LIN {X 0,Y 340.654,Z 947.959,A -85,B 0,C 180,E1 16403.067,E2 16403.067} C_VEL
LIN {X 0,Y 348.105,Z 969.694,A -85,B 0,C 180,E1 16408.833,E2 16408.833} C_VEL
LIN {X 0,Y 350.733,Z 979.844,A -85,B 0,C 180,E1 16411.083,E2 16411.083} C_VEL
LIN {X 0,Y 337.341,Z 1017.391,A -85,B 0,C 180,E1 16414.207,E2 16414.207} C_VEL
LIN {X 0,Y 321.586,Z 1053.328,A -85,B 0,C 180,E1 16418.46,E2 16418.46} C_VEL
LIN {X 0,Y 305.489,Z 1085.768,A -85,B 0,C 180,E1 16424.011,E2 16424.011} C_VEL
LIN {X 0,Y 291.393,Z 1112.806,A -85,B 0,C 180,E1 16430.628,E2 16430.628} C_VEL
LIN {X 0,Y 280.047,Z 1134.815,A -85,B 0,C 180,E1 16438.272,E2 16438.272} C_VEL
LIN {X 0,Y 272.429,Z 1152.316,A -85,B 0,C 180,E1 16447.187,E2 16447.187} C_VEL
LIN {X 0,Y 269.212,Z 1162.751,A -85,B 0,C 180,E1 16455.39,E2 16455.39} C_VEL
LIN {X 0,Y 268.092,Z 1168.645,A -85,B 0,C 180,E1 16463.537,E2 16463.537} C_VEL
LIN {X 0,Y 268.297,Z 1170.082,A -85,B 0,C 180,E1 16470,E2 16470} C_VEL
LIN {X 0,Y 268.113,Z 1168.65,A -85,B 0,C 180,E1 16476.464,E2 16476.464} C_VEL
LIN {X 0,Y 269.134,Z 1162.757,A -85,B 0,C 180,E1 16484.615,E2 16484.615} C_VEL
LIN {X 0,Y 272.422,Z 1152.335,A -85,B 0,C 180,E1 16492.815,E2 16492.815} C_VEL
LIN {X 0,Y 280.074,Z 1134.846,A -85,B 0,C 180,E1 16501.724,E2 16501.724} C_VEL
LIN {X 0,Y 292.426,Z 1110.76,A -85,B 0,C 180,E1 16509.976,E2 16509.976} C_VEL
LIN {X 0,Y 307.416,Z 1082.201,A -85,B 0,C 180,E1 16516.713,E2 16516.713} C_VEL
LIN {X 0,Y 323.735,Z 1049.016,A -85,B 0,C 180,E1 16522.139,E2 16522.139} C_VEL
LIN {X 0,Y 339.489,Z 1012.268,A -85,B 0,C 180,E1 16526.294,E2 16526.294} C_VEL
LIN {X 0,Y 350.803,Z 979.89,A -85,B 0,C 180,E1 16528.924,E2 16528.924} C_VEL
LIN {X 0,Y 344.157,Z 957.095,A -85,B 0,C 180,E1 16534.344,E2 16534.344} C_VEL
LIN {X 0,Y 344.02,Z 956.717,A -85,B 0,C 180,E1 16534.444,E2 16534.444} C_VEL
LIN {X 0,Y 340.378,Z 952.198,A -85,B 0,C 180,E1 16536.416,E2 16536.416} C_VEL
LIN {X 0,Y 333.985,Z 946.963,A -85,B 0,C 180,E1 16539.918,E2 16539.918} C_VEL
LIN {X 0,Y 328.108,Z 933.13,A -85,B 0,C 180,E1 16545.812,E2 16545.812} C_VEL
LIN {X 0,Y 324.423,Z 925.798,A -85,B 0,C 180,E1 16550.715,E2 16550.715} C_VEL
LIN {X 0,Y 322.252,Z 920.268,A -85,B 0,C 180,E1 16555.972,E2 16555.972} C_VEL
LIN {X 0,Y 322.042,Z 920.226,A -85,B 0,C 180,E1 16564.703,E2 16564.703} C_VEL
LIN {X 0,Y 324.764,Z 927.987,A -85,B 0,C 180,E1 16571.677,E2 16571.677} C_VEL
LIN {X 0,Y 328.984,Z 938.356,A -85,B 0,C 180,E1 16577.355,E2 16577.355} C_VEL
LIN {X 0,Y 334.486,Z 953.605,A -85,B 0,C 180,E1 16583.249,E2 16583.249} C_VEL
LIN {X 0,Y 339.367,Z 971.623,A -85,B 0,C 180,E1 16588.478,E2 16588.478} C_VEL
LIN {X 0,Y 341.727,Z 984.521,A -85,B 0,C 180,E1 16591.625,E2 16591.625} C_VEL
LIN {X 0,Y 326.648,Z 1021.482,A -85,B 0,C 180,E1 16595.426,E2 16595.426} C_VEL
LIN {X 0,Y 310.779,Z 1053.687,A -85,B 0,C 180,E1 16600.114,E2 16600.114} C_VEL
LIN {X 0,Y 295.445,Z 1081.297,A -85,B 0,C 180,E1 16605.785,E2 16605.785} C_VEL
LIN {X 0,Y 281.431,Z 1105.448,A -85,B 0,C 180,E1 16612.899,E2 16612.899} C_VEL
LIN {X 0,Y 270.826,Z 1124.108,A -85,B 0,C 180,E1 16620.821,E2 16620.821} C_VEL
LIN {X 0,Y 263.998,Z 1138.31,A -85,B 0,C 180,E1 16629.942,E2 16629.942} C_VEL
LIN {X 0,Y 261.06,Z 1146.198,A -85,B 0,C 180,E1 16638.325,E2 16638.325} C_VEL
LIN {X 0,Y 260.252,Z 1149.946,A -85,B 0,C 180,E1 16646.676,E2 16646.676} C_VEL
LIN {X 0,Y 260.353,Z 1149.923,A -85,B 0,C 180,E1 16653.322,E2 16653.322} C_VEL
LIN {X 0,Y 261.09,Z 1146.107,A -85,B 0,C 180,E1 16661.701,E2 16661.701} C_VEL
LIN {X 0,Y 264.034,Z 1138.177,A -85,B 0,C 180,E1 16670.054,E2 16670.054} C_VEL
LIN {X 0,Y 270.935,Z 1123.932,A -85,B 0,C 180,E1 16679.166,E2 16679.166} C_VEL
LIN {X 0,Y 282.862,Z 1103.055,A -85,B 0,C 180,E1 16687.843,E2 16687.843} C_VEL
LIN {X 0,Y 297.942,Z 1076.932,A -85,B 0,C 180,E1 16695.159,E2 16695.159} C_VEL
LIN {X 0,Y 314.902,Z 1045.612,A -85,B 0,C 180,E1 16701.132,E2 16701.132} C_VEL
LIN {X 0,Y 331.218,Z 1011.108,A -85,B 0,C 180,E1 16705.666,E2 16705.666} C_VEL
LIN {X 0,Y 341.719,Z 984.7,A -85,B 0,C 180,E1 16708.217,E2 16708.217} C_VEL
LIN {X 0,Y 337.435,Z 964.238,A -85,B 0,C 180,E1 16713.437,E2 16713.437} C_VEL
LIN {X 0,Y 331.773,Z 945.868,A -85,B 0,C 180,E1 16719.361,E2 16719.361} C_VEL
LIN {X 0,Y 326.407,Z 931.853,A -85,B 0,C 180,E1 16725.665,E2 16725.665} C_VEL
LIN {X 0,Y 323.079,Z 924.574,A -85,B 0,C 180,E1 16730.998,E2 16730.998} C_VEL
LIN {X 0,Y 322.055,Z 920.268,A -85,B 0,C 180,E1 16734.623,E2 16734.623} C_VEL
LIN {X 0,Y 321.831,Z 919.955,A -85,B 0,C 180,E1 16743.36,E2 16743.36} C_VEL
LIN {X 0,Y 322.694,Z 921.542,A -85,B 0,C 180,E1 16745.907,E2 16745.907} C_VEL
LIN {X 0,Y 325.815,Z 928.749,A -85,B 0,C 180,E1 16751.564,E2 16751.564} C_VEL
LIN {X 0,Y 330.368,Z 938.469,A -85,B 0,C 180,E1 16756.775,E2 16756.775} C_VEL
LIN {X 0,Y 337.309,Z 955.675,A -85,B 0,C 180,E1 16763.044,E2 16763.044} C_VEL
LIN {X 0,Y 343.984,Z 977.436,A -85,B 0,C 180,E1 16768.852,E2 16768.852} C_VEL
LIN {X 0,Y 345.164,Z 984.629,A -85,B 0,C 180,E1 16770.348,E2 16770.348} C_VEL
LIN {X 0,Y 330.908,Z 1021.712,A -85,B 0,C 180,E1 16773.523,E2 16773.523} C_VEL
LIN {X 0,Y 314.982,Z 1056.2,A -85,B 0,C 180,E1 16777.77,E2 16777.77} C_VEL
LIN {X 0,Y 298.773,Z 1087.349,A -85,B 0,C 180,E1 16783.282,E2 16783.282} C_VEL
LIN {X 0,Y 284.328,Z 1113.711,A -85,B 0,C 180,E1 16789.946,E2 16789.946} C_VEL
LIN {X 0,Y 272.063,Z 1136.394,A -85,B 0,C 180,E1 16798.203,E2 16798.203} C_VEL
LIN {X 0,Y 264.38,Z 1153.254,A -85,B 0,C 180,E1 16807.34,E2 16807.34} C_VEL
LIN {X 0,Y 261.037,Z 1164.056,A -85,B 0,C 180,E1 16816.631,E2 16816.631} C_VEL
LIN {X 0,Y 260.187,Z 1168.346,A -85,B 0,C 180,E1 16823.339,E2 16823.339} C_VEL
LIN {X 0,Y 260.397,Z 1169.786,A -85,B 0,C 180,E1 16830,E2 16830} C_VEL
LIN {X 0,Y 260.207,Z 1168.351,A -85,B 0,C 180,E1 16836.661,E2 16836.661} C_VEL
LIN {X 0,Y 261.337,Z 1162.455,A -85,B 0,C 180,E1 16845.061,E2 16845.061} C_VEL
LIN {X 0,Y 264.897,Z 1152.029,A -85,B 0,C 180,E1 16853.501,E2 16853.501} C_VEL
LIN {X 0,Y 273.056,Z 1134.611,A -85,B 0,C 180,E1 16862.604,E2 16862.604} C_VEL
LIN {X 0,Y 285.699,Z 1111.26,A -85,B 0,C 180,E1 16870.816,E2 16870.816} C_VEL
LIN {X 0,Y 301.193,Z 1083.104,A -85,B 0,C 180,E1 16877.62,E2 16877.62} C_VEL
LIN {X 0,Y 318.243,Z 1049.873,A -85,B 0,C 180,E1 16883.146,E2 16883.146} C_VEL
LIN {X 0,Y 334.398,Z 1013.673,A -85,B 0,C 180,E1 16887.292,E2 16887.292} C_VEL
LIN {X 0,Y 345.374,Z 983.208,A -85,B 0,C 180,E1 16889.856,E2 16889.856} C_VEL
LIN {X 0,Y 339.297,Z 961.193,A -85,B 0,C 180,E1 16895.359,E2 16895.359} C_VEL
LIN {X 0,Y 333.985,Z 946.963,A -85,B 0,C 180,E1 16899.918,E2 16899.918} C_VEL
LIN {X 0,Y 330.79,Z 943.941,A -85,B 0,C 180,E1 16902.054,E2 16902.054} C_VEL
LIN {X 0,Y 325.406,Z 941.02,A -85,B 0,C 180,E1 16905.775,E2 16905.775} C_VEL
LIN {X 0,Y 322.278,Z 933.67,A -85,B 0,C 180,E1 16910.228,E2 16910.228} C_VEL
LIN {X 0,Y 320.307,Z 928.989,A -85,B 0,C 180,E1 16914.593,E2 16914.593} C_VEL
LIN {X 0,Y 319.155,Z 927.085,A -85,B 0,C 180,E1 16920,E2 16920} C_VEL
LIN {X 0,Y 319.864,Z 928.113,A -85,B 0,C 180,E1 16925.414,E2 16925.414} C_VEL
LIN {X 0,Y 322.655,Z 937.222,A -85,B 0,C 180,E1 16932.637,E2 16932.637} C_VEL
LIN {X 0,Y 327.152,Z 949.317,A -85,B 0,C 180,E1 16938.836,E2 16938.836} C_VEL
LIN {X 0,Y 331.99,Z 965.451,A -85,B 0,C 180,E1 16944.622,E2 16944.622} C_VEL
LIN {X 0,Y 336.018,Z 985.699,A -85,B 0,C 180,E1 16950.157,E2 16950.157} C_VEL
LIN {X 0,Y 336.292,Z 988.923,A -85,B 0,C 180,E1 16950.887,E2 16950.887} C_VEL
LIN {X 0,Y 319.803,Z 1026.489,A -85,B 0,C 180,E1 16954.833,E2 16954.833} C_VEL
LIN {X 0,Y 303.201,Z 1058.494,A -85,B 0,C 180,E1 16959.741,E2 16959.741} C_VEL
LIN {X 0,Y 286.434,Z 1087.183,A -85,B 0,C 180,E1 16966.094,E2 16966.094} C_VEL
LIN {X 0,Y 271.46,Z 1111.385,A -85,B 0,C 180,E1 16973.971,E2 16973.971} C_VEL
LIN {X 0,Y 260.716,Z 1129.921,A -85,B 0,C 180,E1 16983.107,E2 16983.107} C_VEL
LIN {X 0,Y 254.827,Z 1142.335,A -85,B 0,C 180,E1 16992.777,E2 16992.777} C_VEL
LIN {X 0,Y 252.919,Z 1147.644,A -85,B 0,C 180,E1 16999.689,E2 16999.689} C_VEL
LIN {X 0,Y 252.363,Z 1150.242,A -85,B 0,C 180,E1 17006.572,E2 17006.572} C_VEL
LIN {X 0,Y 252.455,Z 1150.22,A -85,B 0,C 180,E1 17013.426,E2 17013.426} C_VEL
LIN {X 0,Y 253.258,Z 1146.428,A -85,B 0,C 180,E1 17022.037,E2 17022.037} C_VEL
LIN {X 0,Y 256.456,Z 1138.482,A -85,B 0,C 180,E1 17030.673,E2 17030.673} C_VEL
LIN {X 0,Y 263.849,Z 1124.239,A -85,B 0,C 180,E1 17040.028,E2 17040.028} C_VEL
LIN {X 0,Y 276.468,Z 1103.363,A -85,B 0,C 180,E1 17048.88,E2 17048.88} C_VEL
LIN {X 0,Y 292.297,Z 1077.238,A -85,B 0,C 180,E1 17056.283,E2 17056.283} C_VEL
LIN {X 0,Y 309.42,Z 1046.841,A -85,B 0,C 180,E1 17062.155,E2 17062.155} C_VEL
LIN {X 0,Y 326.738,Z 1011.505,A -85,B 0,C 180,E1 17066.813,E2 17066.813} C_VEL
LIN {X 0,Y 336.383,Z 988.492,A -85,B 0,C 180,E1 17069.046,E2 17069.046} C_VEL
LIN {X 0,Y 332.457,Z 968.245,A -85,B 0,C 180,E1 17074.459,E2 17074.459} C_VEL
LIN {X 0,Y 327.465,Z 950.69,A -85,B 0,C 180,E1 17080.484,E2 17080.484} C_VEL
LIN {X 0,Y 323.03,Z 938.176,A -85,B 0,C 180,E1 17086.493,E2 17086.493} C_VEL
LIN {X 0,Y 320.756,Z 932.535,A -85,B 0,C 180,E1 17090.525,E2 17090.525} C_VEL
LIN {X 0,Y 319.702,Z 927.802,A -85,B 0,C 180,E1 17094.584,E2 17094.584} C_VEL
LIN {X 0,Y 319.375,Z 927.351,A -85,B 0,C 180,E1 17102.708,E2 17102.708} C_VEL
LIN {X 0,Y 320.38,Z 929.773,A -85,B 0,C 180,E1 17106.276,E2 17106.276} C_VEL
LIN {X 0,Y 323.432,Z 937.155,A -85,B 0,C 180,E1 17111.983,E2 17111.983} C_VEL
LIN {X 0,Y 328.649,Z 949.187,A -85,B 0,C 180,E1 17118.055,E2 17118.055} C_VEL
LIN {X 0,Y 334.692,Z 966.317,A -85,B 0,C 180,E1 17123.939,E2 17123.939} C_VEL
LIN {X 0,Y 339.971,Z 986.661,A -85,B 0,C 180,E1 17129.225,E2 17129.225} C_VEL
LIN {X 0,Y 323.818,Z 1027.577,A -85,B 0,C 180,E1 17132.986,E2 17132.986} C_VEL
LIN {X 0,Y 306.824,Z 1062.218,A -85,B 0,C 180,E1 17137.528,E2 17137.528} C_VEL
LIN {X 0,Y 289.537,Z 1093.548,A -85,B 0,C 180,E1 17143.538,E2 17143.538} C_VEL
LIN {X 0,Y 273.838,Z 1120.582,A -85,B 0,C 180,E1 17151.154,E2 17151.154} C_VEL
LIN {X 0,Y 262.582,Z 1140.908,A -85,B 0,C 180,E1 17159.541,E2 17159.541} C_VEL
LIN {X 0,Y 255.421,Z 1156.492,A -85,B 0,C 180,E1 17169.239,E2 17169.239} C_VEL
LIN {X 0,Y 252.877,Z 1165.02,A -85,B 0,C 180,E1 17177.945,E2 17177.945} C_VEL
LIN {X 0,Y 252.31,Z 1169.124,A -85,B 0,C 180,E1 17186.572,E2 17186.572} C_VEL
LIN {X 0,Y 252.414,Z 1169.13,A -85,B 0,C 180,E1 17193.428,E2 17193.428} C_VEL
LIN {X 0,Y 252.841,Z 1165.028,A -85,B 0,C 180,E1 17202.058,E2 17202.058} C_VEL
LIN {X 0,Y 255.459,Z 1156.511,A -85,B 0,C 180,E1 17210.759,E2 17210.759} C_VEL
LIN {X 0,Y 262.588,Z 1140.933,A -85,B 0,C 180,E1 17220.461,E2 17220.461} C_VEL
LIN {X 0,Y 274.794,Z 1118.924,A -85,B 0,C 180,E1 17229.425,E2 17229.425} C_VEL
LIN {X 0,Y 290.186,Z 1092.479,A -85,B 0,C 180,E1 17236.721,E2 17236.721} C_VEL
LIN {X 0,Y 307.961,Z 1060.246,A -85,B 0,C 180,E1 17242.774,E2 17242.774} C_VEL
LIN {X 0,Y 324.403,Z 1026.513,A -85,B 0,C 180,E1 17247.147,E2 17247.147} C_VEL
LIN {X 0,Y 340.055,Z 986.698,A -85,B 0,C 180,E1 17250.783,E2 17250.783} C_VEL
LIN {X 0,Y 334.428,Z 965.278,A -85,B 0,C 180,E1 17256.404,E2 17256.404} C_VEL
LIN {X 0,Y 328.767,Z 949.293,A -85,B 0,C 180,E1 17261.952,E2 17261.952} C_VEL
LIN {X 0,Y 325.406,Z 941.02,A -85,B 0,C 180,E1 17265.775,E2 17265.775} C_VEL
LIN {X 0,Y 322.761,Z 939.591,A -85,B 0,C 180,E1 17268.037,E2 17268.037} C_VEL
LIN {X 0,Y 318.588,Z 939.714,A -85,B 0,C 180,E1 17271.935,E2 17271.935} C_VEL
LIN {X 0,Y 317.017,Z 935.024,A -85,B 0,C 180,E1 17277.272,E2 17277.272} C_VEL
LIN {X 0,Y 317.267,Z 935.833,A -85,B 0,C 180,E1 17285.458,E2 17285.458} C_VEL
LIN {X 0,Y 320.306,Z 946.154,A -85,B 0,C 180,E1 17293.624,E2 17293.624} C_VEL
LIN {X 0,Y 324.782,Z 960.499,A -85,B 0,C 180,E1 17300.312,E2 17300.312} C_VEL
LIN {X 0,Y 328.993,Z 978.168,A -85,B 0,C 180,E1 17306.197,E2 17306.197} C_VEL
LIN {X 0,Y 330.992,Z 992.249,A -85,B 0,C 180,E1 17309.977,E2 17309.977} C_VEL
LIN {X 0,Y 314.846,Z 1027.594,A -85,B 0,C 180,E1 17313.736,E2 17313.736} C_VEL
LIN {X 0,Y 297.457,Z 1059.832,A -85,B 0,C 180,E1 17318.741,E2 17318.741} C_VEL
LIN {X 0,Y 280.384,Z 1087.831,A -85,B 0,C 180,E1 17325.031,E2 17325.031} C_VEL
LIN {X 0,Y 264.653,Z 1112.082,A -85,B 0,C 180,E1 17333.104,E2 17333.104} C_VEL
LIN {X 0,Y 254.043,Z 1129.176,A -85,B 0,C 180,E1 17341.627,E2 17341.627} C_VEL
LIN {X 0,Y 247.593,Z 1141.56,A -85,B 0,C 180,E1 17351.184,E2 17351.184} C_VEL
LIN {X 0,Y 244.849,Z 1148.436,A -85,B 0,C 180,E1 17360.416,E2 17360.416} C_VEL
LIN {X 0,Y 244.459,Z 1150.539,A -85,B 0,C 180,E1 17366.461,E2 17366.461} C_VEL
LIN {X 0,Y 244.548,Z 1150.517,A -85,B 0,C 180,E1 17373.537,E2 17373.537} C_VEL
LIN {X 0,Y 245.447,Z 1146.728,A -85,B 0,C 180,E1 17382.426,E2 17382.426} C_VEL
LIN {X 0,Y 248.884,Z 1138.787,A -85,B 0,C 180,E1 17391.333,E2 17391.333} C_VEL
LIN {X 0,Y 256.817,Z 1124.546,A -85,B 0,C 180,E1 17400.939,E2 17400.939} C_VEL
LIN {X 0,Y 270.141,Z 1103.672,A -85,B 0,C 180,E1 17409.97,E2 17409.97} C_VEL
LIN {X 0,Y 286.745,Z 1077.545,A -85,B 0,C 180,E1 17417.456,E2 17417.456} C_VEL
LIN {X 0,Y 304.591,Z 1047.019,A -85,B 0,C 180,E1 17423.377,E2 17423.377} C_VEL
LIN {X 0,Y 322.379,Z 1011.831,A -85,B 0,C 180,E1 17428.013,E2 17428.013} C_VEL
LIN {X 0,Y 330.937,Z 991.647,A -85,B 0,C 180,E1 17430.039,E2 17430.039} C_VEL
LIN {X 0,Y 327.59,Z 972.257,A -85,B 0,C 180,E1 17435.509,E2 17435.509} C_VEL
LIN {X 0,Y 323.199,Z 955.405,A -85,B 0,C 180,E1 17441.609,E2 17441.609} C_VEL
LIN {X 0,Y 319.015,Z 942.705,A -85,B 0,C 180,E1 17448.403,E2 17448.403} C_VEL
LIN {X 0,Y 317.124,Z 935.465,A -85,B 0,C 180,E1 17454.539,E2 17454.539} C_VEL
LIN {X 0,Y 316.841,Z 934.859,A -85,B 0,C 180,E1 17462.73,E2 17462.73} C_VEL
LIN {X 0,Y 317.795,Z 937.468,A -85,B 0,C 180,E1 17466.327,E2 17466.327} C_VEL
LIN {X 0,Y 320.392,Z 944.033,A -85,B 0,C 180,E1 17471.547,E2 17471.547} C_VEL
LIN {X 0,Y 325.044,Z 955.658,A -85,B 0,C 180,E1 17477.563,E2 17477.563} C_VEL
LIN {X 0,Y 330.239,Z 971.625,A -85,B 0,C 180,E1 17483.233,E2 17483.233} C_VEL
LIN {X 0,Y 334.66,Z 990.41,A -85,B 0,C 180,E1 17488.359,E2 17488.359} C_VEL
LIN {X 0,Y 318.845,Z 1028.541,A -85,B 0,C 180,E1 17491.904,E2 17491.904} C_VEL
LIN {X 0,Y 301.916,Z 1061.909,A -85,B 0,C 180,E1 17496.298,E2 17496.298} C_VEL
LIN {X 0,Y 283.646,Z 1093.641,A -85,B 0,C 180,E1 17502.426,E2 17502.426} C_VEL
LIN {X 0,Y 267.263,Z 1120.57,A -85,B 0,C 180,E1 17510.153,E2 17510.153} C_VEL
LIN {X 0,Y 255.257,Z 1141.047,A -85,B 0,C 180,E1 17518.838,E2 17518.838} C_VEL
LIN {X 0,Y 247.821,Z 1156.185,A -85,B 0,C 180,E1 17528.571,E2 17528.571} C_VEL
LIN {X 0,Y 245.039,Z 1164.719,A -85,B 0,C 180,E1 17537.553,E2 17537.553} C_VEL
LIN {X 0,Y 244.397,Z 1168.826,A -85,B 0,C 180,E1 17546.46,E2 17546.46} C_VEL
LIN {X 0,Y 244.496,Z 1168.833,A -85,B 0,C 180,E1 17553.539,E2 17553.539} C_VEL
LIN {X 0,Y 245.002,Z 1164.728,A -85,B 0,C 180,E1 17562.449,E2 17562.449} C_VEL
LIN {X 0,Y 247.847,Z 1156.206,A -85,B 0,C 180,E1 17571.427,E2 17571.427} C_VEL
LIN {X 0,Y 255.258,Z 1141.077,A -85,B 0,C 180,E1 17581.162,E2 17581.162} C_VEL
LIN {X 0,Y 268.149,Z 1119.141,A -85,B 0,C 180,E1 17590.375,E2 17590.375} C_VEL
LIN {X 0,Y 284.581,Z 1092.172,A -85,B 0,C 180,E1 17597.933,E2 17597.933} C_VEL
LIN {X 0,Y 303.072,Z 1059.942,A -85,B 0,C 180,E1 17604.008,E2 17604.008} C_VEL
LIN {X 0,Y 320.18,Z 1026.001,A -85,B 0,C 180,E1 17608.388,E2 17608.388} C_VEL
LIN {X 0,Y 334.728,Z 990.514,A -85,B 0,C 180,E1 17611.643,E2 17611.643} C_VEL
LIN {X 0,Y 329.815,Z 970.026,A -85,B 0,C 180,E1 17617.297,E2 17617.297} C_VEL
LIN {X 0,Y 324.543,Z 954.295,A -85,B 0,C 180,E1 17623.106,E2 17623.106} C_VEL
LIN {X 0,Y 320.123,Z 943.179,A -85,B 0,C 180,E1 17629.132,E2 17629.132} C_VEL
LIN {X 0,Y 318.588,Z 939.714,A -85,B 0,C 180,E1 17631.935,E2 17631.935} C_VEL
LIN {X 0,Y 316.174,Z 940.358,A -85,B 0,C 180,E1 17635.056,E2 17635.056} C_VEL
LIN {X 0,Y 314.142,Z 942.324,A -85,B 0,C 180,E1 17638.241,E2 17638.241} C_VEL
LIN {X 0,Y 314.43,Z 943.479,A -85,B 0,C 180,E1 17645.507,E2 17645.507} C_VEL
LIN {X 0,Y 316.878,Z 952.78,A -85,B 0,C 180,E1 17653.073,E2 17653.073} C_VEL
LIN {X 0,Y 320.69,Z 966.548,A -85,B 0,C 180,E1 17659.761,E2 17659.761} C_VEL
LIN {X 0,Y 324.199,Z 983.558,A -85,B 0,C 180,E1 17665.626,E2 17665.626} C_VEL
LIN {X 0,Y 325.615,Z 995.075,A -85,B 0,C 180,E1 17668.865,E2 17668.865} C_VEL
LIN {X 0,Y 309.543,Z 1029.615,A -85,B 0,C 180,E1 17672.73,E2 17672.73} C_VEL
LIN {X 0,Y 292.457,Z 1060.133,A -85,B 0,C 180,E1 17677.503,E2 17677.503} C_VEL
LIN {X 0,Y 274.51,Z 1088.374,A -85,B 0,C 180,E1 17683.898,E2 17683.898} C_VEL
LIN {X 0,Y 258.206,Z 1112.385,A -85,B 0,C 180,E1 17692.022,E2 17692.022} C_VEL
LIN {X 0,Y 246.894,Z 1129.481,A -85,B 0,C 180,E1 17700.727,E2 17700.727} C_VEL
LIN {X 0,Y 239.975,Z 1141.891,A -85,B 0,C 180,E1 17710.594,E2 17710.594} C_VEL
LIN {X 0,Y 237.235,Z 1148.242,A -85,B 0,C 180,E1 17718.999,E2 17718.999} C_VEL
LIN {X 0,Y 236.574,Z 1150.835,A -85,B 0,C 180,E1 17726.342,E2 17726.342} C_VEL
LIN {X 0,Y 236.656,Z 1150.814,A -85,B 0,C 180,E1 17733.656,E2 17733.656} C_VEL
LIN {X 0,Y 237.645,Z 1147.028,A -85,B 0,C 180,E1 17742.841,E2 17742.841} C_VEL
LIN {X 0,Y 241.353,Z 1139.092,A -85,B 0,C 180,E1 17752.032,E2 17752.032} C_VEL
LIN {X 0,Y 249.703,Z 1125.086,A -85,B 0,C 180,E1 17761.763,E2 17761.763} C_VEL
LIN {X 0,Y 263.954,Z 1103.98,A -85,B 0,C 180,E1 17771.105,E2 17771.105} C_VEL
LIN {X 0,Y 281.331,Z 1077.851,A -85,B 0,C 180,E1 17778.671,E2 17778.671} C_VEL
LIN {X 0,Y 299.85,Z 1047.326,A -85,B 0,C 180,E1 17784.614,E2 17784.614} C_VEL
LIN {X 0,Y 318.376,Z 1011.741,A -85,B 0,C 180,E1 17789.281,E2 17789.281} C_VEL
LIN {X 0,Y 325.548,Z 995.36,A -85,B 0,C 180,E1 17790.95,E2 17790.95} C_VEL
LIN {X 0,Y 322.96,Z 977.426,A -85,B 0,C 180,E1 17796.236,E2 17796.236} C_VEL
LIN {X 0,Y 319.158,Z 961.038,A -85,B 0,C 180,E1 17802.447,E2 17802.447} C_VEL
LIN {X 0,Y 315.806,Z 949.321,A -85,B 0,C 180,E1 17808.982,E2 17808.982} C_VEL
LIN {X 0,Y 314.319,Z 943.078,A -85,B 0,C 180,E1 17814.491,E2 17814.491} C_VEL
LIN {X 0,Y 313.817,Z 941.799,A -85,B 0,C 180,E1 17820,E2 17820} C_VEL
LIN {X 0,Y 314.888,Z 943.933,A -85,B 0,C 180,E1 17825.5,E2 17825.5} C_VEL
LIN {X 0,Y 317.479,Z 951.674,A -85,B 0,C 180,E1 17831.654,E2 17831.654} C_VEL
LIN {X 0,Y 321.628,Z 963.184,A -85,B 0,C 180,E1 17837.566,E2 17837.566} C_VEL
LIN {X 0,Y 326.327,Z 979.643,A -85,B 0,C 180,E1 17843.397,E2 17843.397} C_VEL
LIN {X 0,Y 329.154,Z 995.204,A -85,B 0,C 180,E1 17847.6,E2 17847.6} C_VEL
LIN {X 0,Y 313.372,Z 1030.779,A -85,B 0,C 180,E1 17850.936,E2 17850.936} C_VEL
LIN {X 0,Y 295.985,Z 1063.536,A -85,B 0,C 180,E1 17855.341,E2 17855.341} C_VEL
LIN {X 0,Y 278.137,Z 1093.327,A -85,B 0,C 180,E1 17861.169,E2 17861.169} C_VEL
LIN {X 0,Y 261.446,Z 1119.576,A -85,B 0,C 180,E1 17868.742,E2 17868.742} C_VEL
LIN {X 0,Y 248.137,Z 1140.876,A -85,B 0,C 180,E1 17877.93,E2 17877.93} C_VEL
LIN {X 0,Y 240.251,Z 1155.879,A -85,B 0,C 180,E1 17887.861,E2 17887.861} C_VEL
LIN {X 0,Y 237.196,Z 1164.417,A -85,B 0,C 180,E1 17897.135,E2 17897.135} C_VEL
LIN {X 0,Y 236.509,Z 1168.53,A -85,B 0,C 180,E1 17906.342,E2 17906.342} C_VEL
LIN {X 0,Y 236.599,Z 1168.536,A -85,B 0,C 180,E1 17913.657,E2 17913.657} C_VEL
LIN {X 0,Y 237.154,Z 1164.427,A -85,B 0,C 180,E1 17922.868,E2 17922.868} C_VEL
LIN {X 0,Y 240.267,Z 1155.901,A -85,B 0,C 180,E1 17932.138,E2 17932.138} C_VEL
LIN {X 0,Y 248.14,Z 1140.907,A -85,B 0,C 180,E1 17942.07,E2 17942.07} C_VEL
LIN {X 0,Y 262.074,Z 1118.519,A -85,B 0,C 180,E1 17951.656,E2 17951.656} C_VEL
LIN {X 0,Y 279.131,Z 1091.865,A -85,B 0,C 180,E1 17959.188,E2 17959.188} C_VEL
LIN {X 0,Y 298.177,Z 1059.96,A -85,B 0,C 180,E1 17965.228,E2 17965.228} C_VEL
LIN {X 0,Y 315.978,Z 1025.7,A -85,B 0,C 180,E1 17969.649,E2 17969.649} C_VEL
LIN {X 0,Y 329.442,Z 994.206,A -85,B 0,C 180,E1 17972.555,E2 17972.555} C_VEL
LIN {X 0,Y 325.186,Z 974.672,A -85,B 0,C 180,E1 17978.209,E2 17978.209} C_VEL
LIN {X 0,Y 319.941,Z 957.714,A -85,B 0,C 180,E1 17984.965,E2 17984.965} C_VEL
LIN {X 0,Y 316.604,Z 948.591,A -85,B 0,C 180,E1 17990.397,E2 17990.397} C_VEL
LIN {X 0,Y 314.365,Z 942.501,A -85,B 0,C 180,E1 17997.248,E2 17997.248} C_VEL
LIN {X 0,Y 314.142,Z 942.324,A -85,B 0,C 180,E1 17998.241,E2 17998.241} C_VEL
LIN {X 0,Y 312.98,Z 944.5,A -85,B 0,C 180,E1 18000.591,E2 18000.591} C_VEL
LIN {X 0,Y 311.27,Z 950.531,A -85,B 0,C 180,E1 18004.486,E2 18004.486} C_VEL
LIN {X 0,Y 313.002,Z 958.355,A -85,B 0,C 180,E1 18011.862,E2 18011.862} C_VEL
LIN {X 0,Y 315.902,Z 969.965,A -85,B 0,C 180,E1 18018.087,E2 18018.087} C_VEL
LIN {X 0,Y 318.897,Z 985.147,A -85,B 0,C 180,E1 18023.854,E2 18023.854} C_VEL
LIN {X 0,Y 320.402,Z 999.386,A -85,B 0,C 180,E1 18028.096,E2 18028.096} C_VEL
LIN {X 0,Y 302.064,Z 1035.805,A -85,B 0,C 180,E1 18032.238,E2 18032.238} C_VEL
LIN {X 0,Y 282.736,Z 1068.06,A -85,B 0,C 180,E1 18037.717,E2 18037.717} C_VEL
LIN {X 0,Y 263.636,Z 1096.281,A -85,B 0,C 180,E1 18044.901,E2 18044.901} C_VEL
LIN {X 0,Y 247.602,Z 1118.601,A -85,B 0,C 180,E1 18053.543,E2 18053.543} C_VEL
LIN {X 0,Y 236.514,Z 1135.046,A -85,B 0,C 180,E1 18063.473,E2 18063.473} C_VEL
LIN {X 0,Y 231.074,Z 1144.746,A -85,B 0,C 180,E1 18072.91,E2 18072.91} C_VEL
LIN {X 0,Y 228.826,Z 1150.169,A -85,B 0,C 180,E1 18082.421,E2 18082.421} C_VEL
LIN {X 0,Y 228.826,Z 1151.439,A -85,B 0,C 180,E1 18090,E2 18090} C_VEL
LIN {X 0,Y 228.928,Z 1149.685,A -85,B 0,C 180,E1 18098.621,E2 18098.621} C_VEL
LIN {X 0,Y 231.908,Z 1143.138,A -85,B 0,C 180,E1 18108.986,E2 18108.986} C_VEL
LIN {X 0,Y 239.023,Z 1131.006,A -85,B 0,C 180,E1 18119.306,E2 18119.306} C_VEL
LIN {X 0,Y 251.683,Z 1112.836,A -85,B 0,C 180,E1 18128.942,E2 18128.942} C_VEL
LIN {X 0,Y 269.18,Z 1088.224,A -85,B 0,C 180,E1 18137.372,E2 18137.372} C_VEL
LIN {X 0,Y 288.831,Z 1058.275,A -85,B 0,C 180,E1 18144.076,E2 18144.076} C_VEL
LIN {X 0,Y 307.975,Z 1024.808,A -85,B 0,C 180,E1 18149.066,E2 18149.066} C_VEL
LIN {X 0,Y 320.284,Z 999.009,A -85,B 0,C 180,E1 18151.893,E2 18151.893} C_VEL
LIN {X 0,Y 317.93,Z 980.405,A -85,B 0,C 180,E1 18157.686,E2 18157.686} C_VEL
LIN {X 0,Y 314.784,Z 965.345,A -85,B 0,C 180,E1 18163.928,E2 18163.928} C_VEL
LIN {X 0,Y 312.153,Z 955.119,A -85,B 0,C 180,E1 18170.259,E2 18170.259} C_VEL
LIN {X 0,Y 311.384,Z 950.653,A -85,B 0,C 180,E1 18174.438,E2 18174.438} C_VEL
LIN {X 0,Y 310.96,Z 949.138,A -85,B 0,C 180,E1 18180,E2 18180} C_VEL
LIN {X 0,Y 311.957,Z 951.499,A -85,B 0,C 180,E1 18185.552,E2 18185.552} C_VEL
LIN {X 0,Y 314.837,Z 960.262,A -85,B 0,C 180,E1 18192.455,E2 18192.455} C_VEL
LIN {X 0,Y 319.301,Z 975.052,A -85,B 0,C 180,E1 18199.318,E2 18199.318} C_VEL
LIN {X 0,Y 323.284,Z 993.187,A -85,B 0,C 180,E1 18205.205,E2 18205.205} C_VEL
LIN {X 0,Y 323.828,Z 999.031,A -85,B 0,C 180,E1 18206.653,E2 18206.653} C_VEL
LIN {X 0,Y 306.067,Z 1036.835,A -85,B 0,C 180,E1 18210.367,E2 18210.367} C_VEL
LIN {X 0,Y 286.486,Z 1071.386,A -85,B 0,C 180,E1 18215.407,E2 18215.407} C_VEL
LIN {X 0,Y 267.006,Z 1101.874,A -85,B 0,C 180,E1 18222.118,E2 18222.118} C_VEL
LIN {X 0,Y 249.734,Z 1127.363,A -85,B 0,C 180,E1 18230.62,E2 18230.62} C_VEL
LIN {X 0,Y 237.469,Z 1146.646,A -85,B 0,C 180,E1 18240.497,E2 18240.497} C_VEL
LIN {X 0,Y 230.945,Z 1159.588,A -85,B 0,C 180,E1 18250.932,E2 18250.932} C_VEL
LIN {X 0,Y 229.033,Z 1165.361,A -85,B 0,C 180,E1 18258.6,E2 18258.6} C_VEL
LIN {X 0,Y 228.593,Z 1168.232,A -85,B 0,C 180,E1 18266.215,E2 18266.215} C_VEL
LIN {X 0,Y 228.679,Z 1168.239,A -85,B 0,C 180,E1 18273.784,E2 18273.784} C_VEL
LIN {X 0,Y 229.317,Z 1164.125,A -85,B 0,C 180,E1 18283.316,E2 18283.316} C_VEL
LIN {X 0,Y 232.71,Z 1155.595,A -85,B 0,C 180,E1 18292.897,E2 18292.897} C_VEL
LIN {X 0,Y 241.308,Z 1140.386,A -85,B 0,C 180,E1 18303.236,E2 18303.236} C_VEL
LIN {X 0,Y 255.557,Z 1118.818,A -85,B 0,C 180,E1 18312.679,E2 18312.679} C_VEL
LIN {X 0,Y 273.777,Z 1091.557,A -85,B 0,C 180,E1 18320.503,E2 18320.503} C_VEL
LIN {X 0,Y 293.361,Z 1060.06,A -85,B 0,C 180,E1 18326.48,E2 18326.48} C_VEL
LIN {X 0,Y 312.039,Z 1025.234,A -85,B 0,C 180,E1 18330.952,E2 18330.952} C_VEL
LIN {X 0,Y 323.911,Z 999.033,A -85,B 0,C 180,E1 18333.369,E2 18333.369} C_VEL
LIN {X 0,Y 321.61,Z 984.038,A -85,B 0,C 180,E1 18337.591,E2 18337.591} C_VEL
LIN {X 0,Y 317.518,Z 968.509,A -85,B 0,C 180,E1 18343.432,E2 18343.432} C_VEL
LIN {X 0,Y 313.833,Z 957.426,A -85,B 0,C 180,E1 18349.612,E2 18349.612} C_VEL
LIN {X 0,Y 312.044,Z 951.839,A -85,B 0,C 180,E1 18354.45,E2 18354.45} C_VEL
LIN {X 0,Y 311.117,Z 949.362,A -85,B 0,C 180,E1 18360,E2 18360} C_VEL
LIN {X 0,Y 311.27,Z 950.531,A -85,B 0,C 180,E1 18364.486,E2 18364.486} C_VEL
LIN {X 0,Y 310.666,Z 954.462,A -85,B 0,C 180,E1 18366.781,E2 18366.781} C_VEL
LIN {X 0,Y 309.21,Z 963.811,A -85,B 0,C 180,E1 18370.499,E2 18370.499} C_VEL
LIN {X 0,Y 311.527,Z 974.688,A -85,B 0,C 180,E1 18376.895,E2 18376.895} C_VEL
LIN {X 0,Y 314.143,Z 989.887,A -85,B 0,C 180,E1 18383.018,E2 18383.018} C_VEL
LIN {X 0,Y 314.895,Z 1003.676,A -85,B 0,C 180,E1 18387.214,E2 18387.214} C_VEL
LIN {X 0,Y 296.033,Z 1039.252,A -85,B 0,C 180,E1 18391.369,E2 18391.369} C_VEL
LIN {X 0,Y 275.946,Z 1071.153,A -85,B 0,C 180,E1 18396.978,E2 18396.978} C_VEL
LIN {X 0,Y 257.026,Z 1097.797,A -85,B 0,C 180,E1 18404.011,E2 18404.011} C_VEL
LIN {X 0,Y 241.062,Z 1118.906,A -85,B 0,C 180,E1 18412.386,E2 18412.386} C_VEL
LIN {X 0,Y 229.267,Z 1135.349,A -85,B 0,C 180,E1 18422.565,E2 18422.565} C_VEL
LIN {X 0,Y 223.381,Z 1145.065,A -85,B 0,C 180,E1 18432.326,E2 18432.326} C_VEL
LIN {X 0,Y 220.952,Z 1150.467,A -85,B 0,C 180,E1 18442.149,E2 18442.149} C_VEL
LIN {X 0,Y 220.951,Z 1151.735,A -85,B 0,C 180,E1 18450,E2 18450} C_VEL
LIN {X 0,Y 220.978,Z 1150.429,A -85,B 0,C 180,E1 18457.849,E2 18457.849} C_VEL
LIN {X 0,Y 223.41,Z 1144.963,A -85,B 0,C 180,E1 18467.695,E2 18467.695} C_VEL
LIN {X 0,Y 229.287,Z 1135.206,A -85,B 0,C 180,E1 18477.431,E2 18477.431} C_VEL
LIN {X 0,Y 241.199,Z 1118.706,A -85,B 0,C 180,E1 18487.588,E2 18487.588} C_VEL
LIN {X 0,Y 258.06,Z 1096.315,A -85,B 0,C 180,E1 18496.355,E2 18496.355} C_VEL
LIN {X 0,Y 277.605,Z 1068.612,A -85,B 0,C 180,E1 18503.443,E2 18503.443} C_VEL
LIN {X 0,Y 297.475,Z 1036.67,A -85,B 0,C 180,E1 18508.873,E2 18508.873} C_VEL
LIN {X 0,Y 315.047,Z 1002.745,A -85,B 0,C 180,E1 18512.842,E2 18512.842} C_VEL
LIN {X 0,Y 313.149,Z 984.54,A -85,B 0,C 180,E1 18518.814,E2 18518.814} C_VEL
LIN {X 0,Y 310.565,Z 970.237,A -85,B 0,C 180,E1 18525.15,E2 18525.15} C_VEL
LIN {X 0,Y 308.468,Z 961.116,A -85,B 0,C 180,E1 18531.561,E2 18531.561} C_VEL
LIN {X 0,Y 308.193,Z 958.115,A -85,B 0,C 180,E1 18534.381,E2 18534.381} C_VEL
LIN {X 0,Y 307.964,Z 956.444,A -85,B 0,C 180,E1 18540,E2 18540} C_VEL
LIN {X 0,Y 308.837,Z 958.969,A -85,B 0,C 180,E1 18545.608,E2 18545.608} C_VEL
LIN {X 0,Y 311.469,Z 967.62,A -85,B 0,C 180,E1 18552.437,E2 18552.437} C_VEL
LIN {X 0,Y 315.256,Z 981.845,A -85,B 0,C 180,E1 18559.102,E2 18559.102} C_VEL
LIN {X 0,Y 318.549,Z 999.487,A -85,B 0,C 180,E1 18564.91,E2 18564.91} C_VEL
LIN {X 0,Y 318.239,Z 1003.216,A -85,B 0,C 180,E1 18565.719,E2 18565.719} C_VEL
LIN {X 0,Y 300.72,Z 1038.92,A -85,B 0,C 180,E1 18569.323,E2 18569.323} C_VEL
LIN {X 0,Y 281.004,Z 1072.329,A -85,B 0,C 180,E1 18574.273,E2 18574.273} C_VEL
LIN {X 0,Y 261.544,Z 1101.579,A -85,B 0,C 180,E1 18580.784,E2 18580.784} C_VEL
LIN {X 0,Y 243.382,Z 1127.05,A -85,B 0,C 180,E1 18589.382,E2 18589.382} C_VEL
LIN {X 0,Y 230.321,Z 1146.336,A -85,B 0,C 180,E1 18599.485,E2 18599.485} C_VEL
LIN {X 0,Y 223.262,Z 1159.282,A -85,B 0,C 180,E1 18610.249,E2 18610.249} C_VEL
LIN {X 0,Y 221.179,Z 1165.06,A -85,B 0,C 180,E1 18618.19,E2 18618.19} C_VEL
LIN {X 0,Y 220.683,Z 1167.935,A -85,B 0,C 180,E1 18626.08,E2 18626.08} C_VEL
LIN {X 0,Y 220.94,Z 1168.306,A -85,B 0,C 180,E1 18630,E2 18630} C_VEL
LIN {X 0,Y 220.723,Z 1166.86,A -85,B 0,C 180,E1 18637.859,E2 18637.859} C_VEL
LIN {X 0,Y 222.362,Z 1161.446,A -85,B 0,C 180,E1 18647.149,E2 18647.149} C_VEL
LIN {X 0,Y 227.857,Z 1150.495,A -85,B 0,C 180,E1 18657.619,E2 18657.619} C_VEL
LIN {X 0,Y 239.703,Z 1132.405,A -85,B 0,C 180,E1 18668.247,E2 18668.247} C_VEL
LIN {X 0,Y 255.496,Z 1110.138,A -85,B 0,C 180,E1 18676.766,E2 18676.766} C_VEL
LIN {X 0,Y 275.18,Z 1081.488,A -85,B 0,C 180,E1 18683.984,E2 18683.984} C_VEL
LIN {X 0,Y 295.785,Z 1047.842,A -85,B 0,C 180,E1 18689.58,E2 18689.58} C_VEL
LIN {X 0,Y 315.244,Z 1010.18,A -85,B 0,C 180,E1 18693.694,E2 18693.694} C_VEL
LIN {X 0,Y 318.913,Z 1001.418,A -85,B 0,C 180,E1 18694.537,E2 18694.537} C_VEL
LIN {X 0,Y 315.652,Z 983.151,A -85,B 0,C 180,E1 18700.45,E2 18700.45} C_VEL
LIN {X 0,Y 312.023,Z 969.214,A -85,B 0,C 180,E1 18706.749,E2 18706.749} C_VEL
LIN {X 0,Y 309.315,Z 961.136,A -85,B 0,C 180,E1 18712.648,E2 18712.648} C_VEL
LIN {X 0,Y 308.46,Z 957.259,A -85,B 0,C 180,E1 18717.196,E2 18717.196} C_VEL
LIN {X 0,Y 308.073,Z 957.028,A -85,B 0,C 180,E1 18722.807,E2 18722.807} C_VEL
LIN {X 0,Y 308.345,Z 960.034,A -85,B 0,C 180,E1 18727.064,E2 18727.064} C_VEL
LIN {X 0,Y 309.21,Z 963.811,A -85,B 0,C 180,E1 18730.499,E2 18730.499} C_VEL
LIN {X 0,Y 308.742,Z 969.359,A -85,B 0,C 180,E1 18732.705,E2 18732.705} C_VEL
LIN {X 0,Y 307.354,Z 980.591,A -85,B 0,C 180,E1 18736.258,E2 18736.258} C_VEL
LIN {X 0,Y 309.322,Z 995.398,A -85,B 0,C 180,E1 18742.467,E2 18742.467} C_VEL
LIN {X 0,Y 309.65,Z 1007.266,A -85,B 0,C 180,E1 18746.226,E2 18746.226} C_VEL
LIN {X 0,Y 291.282,Z 1040.584,A -85,B 0,C 180,E1 18750.172,E2 18750.172} C_VEL
LIN {X 0,Y 271.167,Z 1071.453,A -85,B 0,C 180,E1 18755.615,E2 18755.615} C_VEL
LIN {X 0,Y 251.436,Z 1098.1,A -85,B 0,C 180,E1 18762.676,E2 18762.676} C_VEL
LIN {X 0,Y 234.632,Z 1119.212,A -85,B 0,C 180,E1 18771.166,E2 18771.166} C_VEL
LIN {X 0,Y 222.085,Z 1135.653,A -85,B 0,C 180,E1 18781.599,E2 18781.599} C_VEL
LIN {X 0,Y 215.664,Z 1145.501,A -85,B 0,C 180,E1 18791.863,E2 18791.863} C_VEL
LIN {X 0,Y 213.105,Z 1150.764,A -85,B 0,C 180,E1 18801.858,E2 18801.858} C_VEL
LIN {X 0,Y 213.049,Z 1152.031,A -85,B 0,C 180,E1 18810,E2 18810} C_VEL
LIN {X 0,Y 213.118,Z 1150.727,A -85,B 0,C 180,E1 18818.141,E2 18818.141} C_VEL
LIN {X 0,Y 215.693,Z 1145.404,A -85,B 0,C 180,E1 18828.153,E2 18828.153} C_VEL
LIN {X 0,Y 222.106,Z 1135.512,A -85,B 0,C 180,E1 18838.397,E2 18838.397} C_VEL
LIN {X 0,Y 234.767,Z 1119.014,A -85,B 0,C 180,E1 18848.807,E2 18848.807} C_VEL
LIN {X 0,Y 252.493,Z 1096.623,A -85,B 0,C 180,E1 18857.696,E2 18857.696} C_VEL
LIN {X 0,Y 272.863,Z 1068.916,A -85,B 0,C 180,E1 18864.81,E2 18864.81} C_VEL
LIN {X 0,Y 293.393,Z 1036.976,A -85,B 0,C 180,E1 18870.219,E2 18870.219} C_VEL
LIN {X 0,Y 309.649,Z 1006.97,A -85,B 0,C 180,E1 18873.706,E2 18873.706} C_VEL
LIN {X 0,Y 308.622,Z 989.889,A -85,B 0,C 180,E1 18879.523,E2 18879.523} C_VEL
LIN {X 0,Y 306.623,Z 976.416,A -85,B 0,C 180,E1 18885.756,E2 18885.756} C_VEL
LIN {X 0,Y 304.967,Z 967.417,A -85,B 0,C 180,E1 18892.491,E2 18892.491} C_VEL
LIN {X 0,Y 304.704,Z 964.081,A -85,B 0,C 180,E1 18897.162,E2 18897.162} C_VEL
LIN {X 0,Y 305.083,Z 964.38,A -85,B 0,C 180,E1 18902.835,E2 18902.835} C_VEL
LIN {X 0,Y 306.862,Z 971.106,A -85,B 0,C 180,E1 18909.912,E2 18909.912} C_VEL
LIN {X 0,Y 309.714,Z 982.391,A -85,B 0,C 180,E1 18916.268,E2 18916.268} C_VEL
LIN {X 0,Y 312.596,Z 997.479,A -85,B 0,C 180,E1 18922.07,E2 18922.07} C_VEL
LIN {X 0,Y 313.163,Z 1006.489,A -85,B 0,C 180,E1 18924.695,E2 18924.695} C_VEL
LIN {X 0,Y 295.37,Z 1041.117,A -85,B 0,C 180,E1 18928.264,E2 18928.264} C_VEL
LIN {X 0,Y 276.208,Z 1072.433,A -85,B 0,C 180,E1 18932.953,E2 18932.953} C_VEL
LIN {X 0,Y 256.13,Z 1101.374,A -85,B 0,C 180,E1 18939.412,E2 18939.412} C_VEL
LIN {X 0,Y 237.179,Z 1126.74,A -85,B 0,C 180,E1 18948.084,E2 18948.084} C_VEL
LIN {X 0,Y 223.264,Z 1146.026,A -85,B 0,C 180,E1 18958.412,E2 18958.412} C_VEL
LIN {X 0,Y 215.612,Z 1158.976,A -85,B 0,C 180,E1 18969.517,E2 18969.517} C_VEL
LIN {X 0,Y 213.335,Z 1164.759,A -85,B 0,C 180,E1 18977.749,E2 18977.749} C_VEL
LIN {X 0,Y 212.767,Z 1167.637,A -85,B 0,C 180,E1 18985.933,E2 18985.933} C_VEL
LIN {X 0,Y 213.035,Z 1168.01,A -85,B 0,C 180,E1 18990,E2 18990} C_VEL
LIN {X 0,Y 212.823,Z 1166.561,A -85,B 0,C 180,E1 18998.153,E2 18998.153} C_VEL
LIN {X 0,Y 214.178,Z 1162.251,A -85,B 0,C 180,E1 19006.37,E2 19006.37} C_VEL
LIN {X 0,Y 219.632,Z 1151.738,A -85,B 0,C 180,E1 19017.346,E2 19017.346} C_VEL
LIN {X 0,Y 231.218,Z 1134.839,A -85,B 0,C 180,E1 19028.136,E2 19028.136} C_VEL
LIN {X 0,Y 247.35,Z 1113.122,A -85,B 0,C 180,E1 19037.062,E2 19037.062} C_VEL
LIN {X 0,Y 265.849,Z 1087.705,A -85,B 0,C 180,E1 19043.985,E2 19043.985} C_VEL
LIN {X 0,Y 285.614,Z 1057.786,A -85,B 0,C 180,E1 19049.484,E2 19049.484} C_VEL
LIN {X 0,Y 305.435,Z 1022.745,A -85,B 0,C 180,E1 19053.806,E2 19053.806} C_VEL
LIN {X 0,Y 313.668,Z 1005.05,A -85,B 0,C 180,E1 19055.547,E2 19055.547} C_VEL
LIN {X 0,Y 310.867,Z 987.501,A -85,B 0,C 180,E1 19061.608,E2 19061.608} C_VEL
LIN {X 0,Y 307.777,Z 974.384,A -85,B 0,C 180,E1 19068.003,E2 19068.003} C_VEL
LIN {X 0,Y 305.673,Z 966.652,A -85,B 0,C 180,E1 19074.334,E2 19074.334} C_VEL
LIN {X 0,Y 305.252,Z 964.519,A -85,B 0,C 180,E1 19077.166,E2 19077.166} C_VEL
LIN {X 0,Y 304.868,Z 964.282,A -85,B 0,C 180,E1 19082.837,E2 19082.837} C_VEL
LIN {X 0,Y 305.263,Z 968.845,A -85,B 0,C 180,E1 19088.633,E2 19088.633} C_VEL
LIN {X 0,Y 306.981,Z 978.092,A -85,B 0,C 180,E1 19094.955,E2 19094.955} C_VEL
LIN {X 0,Y 307.354,Z 980.591,A -85,B 0,C 180,E1 19096.258,E2 19096.258} C_VEL
LIN {X 0,Y 306.817,Z 987.262,A -85,B 0,C 180,E1 19098.366,E2 19098.366} C_VEL
LIN {X 0,Y 304.479,Z 1000.395,A -85,B 0,C 180,E1 19101.704,E2 19101.704} C_VEL
LIN {X 0,Y 304.226,Z 1011.378,A -85,B 0,C 180,E1 19105.253,E2 19105.253} C_VEL
LIN {X 0,Y 284.692,Z 1045.019,A -85,B 0,C 180,E1 19109.392,E2 19109.392} C_VEL
LIN {X 0,Y 264.46,Z 1074.467,A -85,B 0,C 180,E1 19114.79,E2 19114.79} C_VEL
LIN {X 0,Y 244.977,Z 1099.594,A -85,B 0,C 180,E1 19121.688,E2 19121.688} C_VEL
LIN {X 0,Y 228.332,Z 1119.516,A -85,B 0,C 180,E1 19129.881,E2 19129.881} C_VEL
LIN {X 0,Y 214.947,Z 1135.958,A -85,B 0,C 180,E1 19140.565,E2 19140.565} C_VEL
LIN {X 0,Y 207.841,Z 1146.132,A -85,B 0,C 180,E1 19151.638,E2 19151.638} C_VEL
LIN {X 0,Y 205.23,Z 1151.062,A -85,B 0,C 180,E1 19161.543,E2 19161.543} C_VEL
LIN {X 0,Y 205.149,Z 1152.327,A -85,B 0,C 180,E1 19170,E2 19170} C_VEL
LIN {X 0,Y 205.244,Z 1151.026,A -85,B 0,C 180,E1 19178.455,E2 19178.455} C_VEL
LIN {X 0,Y 208.5,Z 1145.021,A -85,B 0,C 180,E1 19189.809,E2 19189.809} C_VEL
LIN {X 0,Y 215.918,Z 1134.527,A -85,B 0,C 180,E1 19200.443,E2 19200.443} C_VEL
LIN {X 0,Y 228.476,Z 1119.322,A -85,B 0,C 180,E1 19210.087,E2 19210.087} C_VEL
LIN {X 0,Y 247.039,Z 1096.934,A -85,B 0,C 180,E1 19219.105,E2 19219.105} C_VEL
LIN {X 0,Y 268.035,Z 1069.572,A -85,B 0,C 180,E1 19226.154,E2 19226.154} C_VEL
LIN {X 0,Y 289.489,Z 1037.281,A -85,B 0,C 180,E1 19231.598,E2 19231.598} C_VEL
LIN {X 0,Y 304.21,Z 1011.096,A -85,B 0,C 180,E1 19234.68,E2 19234.68} C_VEL
LIN {X 0,Y 304.093,Z 997.776,A -85,B 0,C 180,E1 19239.204,E2 19239.204} C_VEL
LIN {X 0,Y 302.693,Z 983.901,A -85,B 0,C 180,E1 19245.567,E2 19245.567} C_VEL
LIN {X 0,Y 301.541,Z 975.707,A -85,B 0,C 180,E1 19251.366,E2 19251.366} C_VEL
LIN {X 0,Y 301.299,Z 971.24,A -85,B 0,C 180,E1 19257.13,E2 19257.13} C_VEL
LIN {X 0,Y 301.697,Z 971.595,A -85,B 0,C 180,E1 19262.867,E2 19262.867} C_VEL
LIN {X 0,Y 303.248,Z 978.482,A -85,B 0,C 180,E1 19270.031,E2 19270.031} C_VEL
LIN {X 0,Y 305.447,Z 988.486,A -85,B 0,C 180,E1 19275.766,E2 19275.766} C_VEL
LIN {X 0,Y 307.758,Z 1003.101,A -85,B 0,C 180,E1 19281.574,E2 19281.574} C_VEL
LIN {X 0,Y 308.348,Z 1009.44,A -85,B 0,C 180,E1 19283.613,E2 19283.613} C_VEL
LIN {X 0,Y 288.958,Z 1045.264,A -85,B 0,C 180,E1 19287.405,E2 19287.405} C_VEL
LIN {X 0,Y 269.368,Z 1075.592,A -85,B 0,C 180,E1 19292.145,E2 19292.145} C_VEL
LIN {X 0,Y 248.913,Z 1103.688,A -85,B 0,C 180,E1 19298.718,E2 19298.718} C_VEL
LIN {X 0,Y 230.874,Z 1126.683,A -85,B 0,C 180,E1 19306.828,E2 19306.828} C_VEL
LIN {X 0,Y 216.077,Z 1145.984,A -85,B 0,C 180,E1 19317.464,E2 19317.464} C_VEL
LIN {X 0,Y 208.021,Z 1158.671,A -85,B 0,C 180,E1 19328.734,E2 19328.734} C_VEL
LIN {X 0,Y 205.501,Z 1164.457,A -85,B 0,C 180,E1 19337.274,E2 19337.274} C_VEL
LIN {X 0,Y 204.865,Z 1167.34,A -85,B 0,C 180,E1 19345.776,E2 19345.776} C_VEL
LIN {X 0,Y 205.134,Z 1167.714,A -85,B 0,C 180,E1 19350,E2 19350} C_VEL
LIN {X 0,Y 204.925,Z 1166.262,A -85,B 0,C 180,E1 19358.469,E2 19358.469} C_VEL
LIN {X 0,Y 206.939,Z 1160.766,A -85,B 0,C 180,E1 19368.569,E2 19368.569} C_VEL
LIN {X 0,Y 213.431,Z 1149.881,A -85,B 0,C 180,E1 19379.665,E2 19379.665} C_VEL
LIN {X 0,Y 226.747,Z 1131.987,A -85,B 0,C 180,E1 19390.748,E2 19390.748} C_VEL
LIN {X 0,Y 245.621,Z 1108.006,A -85,B 0,C 180,E1 19400.044,E2 19400.044} C_VEL
LIN {X 0,Y 265.84,Z 1080.877,A -85,B 0,C 180,E1 19406.854,E2 19406.854} C_VEL
LIN {X 0,Y 287.252,Z 1048.274,A -85,B 0,C 180,E1 19412.253,E2 19412.253} C_VEL
LIN {X 0,Y 307.773,Z 1010.93,A -85,B 0,C 180,E1 19416.28,E2 19416.28} C_VEL
LIN {X 0,Y 308.333,Z 1007.659,A -85,B 0,C 180,E1 19416.951,E2 19416.951} C_VEL
LIN {X 0,Y 306.134,Z 991.814,A -85,B 0,C 180,E1 19422.798,E2 19422.798} C_VEL
LIN {X 0,Y 303.875,Z 980.752,A -85,B 0,C 180,E1 19428.543,E2 19428.543} C_VEL
LIN {X 0,Y 301.98,Z 972.714,A -85,B 0,C 180,E1 19435.701,E2 19435.701} C_VEL
LIN {X 0,Y 301.561,Z 971.018,A -85,B 0,C 180,E1 19440,E2 19440} C_VEL
LIN {X 0,Y 301.488,Z 973.099,A -85,B 0,C 180,E1 19445.745,E2 19445.745} C_VEL
LIN {X 0,Y 302.525,Z 981.72,A -85,B 0,C 180,E1 19452.97,E2 19452.97} C_VEL
LIN {X 0,Y 304.122,Z 995.702,A -85,B 0,C 180,E1 19459.883,E2 19459.883} C_VEL
LIN {X 0,Y 304.479,Z 1000.395,A -85,B 0,C 180,E1 19461.704,E2 19461.704} C_VEL
LIN {X 0,Y 302.923,Z 1007.199,A -85,B 0,C 180,E1 19463.258,E2 19463.258} C_VEL
LIN {X 0,Y 296.689,Z 1019.647,A -85,B 0,C 180,E1 19464.74,E2 19464.74} C_VEL
LIN {X 0,Y 292.357,Z 1026.918,A -85,B 0,C 180,E1 19465.516,E2 19465.516} C_VEL
LIN {X 0,Y 270.627,Z 1060.407,A -85,B 0,C 180,E1 19470.431,E2 19470.431} C_VEL
LIN {X 0,Y 248.168,Z 1089.714,A -85,B 0,C 180,E1 19477.052,E2 19477.052} C_VEL
LIN {X 0,Y 227.271,Z 1114.126,A -85,B 0,C 180,E1 19485.799,E2 19485.799} C_VEL
LIN {X 0,Y 211.097,Z 1132.388,A -85,B 0,C 180,E1 19496.357,E2 19496.357} C_VEL
LIN {X 0,Y 201.619,Z 1144.446,A -85,B 0,C 180,E1 19508.023,E2 19508.023} C_VEL
LIN {X 0,Y 198.206,Z 1149.736,A -85,B 0,C 180,E1 19516.797,E2 19516.797} C_VEL
LIN {X 0,Y 197.083,Z 1152.319,A -85,B 0,C 180,E1 19525.608,E2 19525.608} C_VEL
LIN {X 0,Y 197.149,Z 1152.3,A -85,B 0,C 180,E1 19534.389,E2 19534.389} C_VEL
LIN {X 0,Y 198.845,Z 1148.531,A -85,B 0,C 180,E1 19545.403,E2 19545.403} C_VEL
LIN {X 0,Y 204.366,Z 1140.616,A -85,B 0,C 180,E1 19556.297,E2 19556.297} C_VEL
LIN {X 0,Y 216.139,Z 1126.638,A -85,B 0,C 180,E1 19567.44,E2 19567.44} C_VEL
LIN {X 0,Y 234.953,Z 1105.254,A -85,B 0,C 180,E1 19577.767,E2 19577.767} C_VEL
LIN {X 0,Y 256.324,Z 1079.389,A -85,B 0,C 180,E1 19585.507,E2 19585.507} C_VEL
LIN {X 0,Y 278.293,Z 1049.062,A -85,B 0,C 180,E1 19591.371,E2 19591.371} C_VEL
LIN {X 0,Y 299.454,Z 1013.654,A -85,B 0,C 180,E1 19595.948,E2 19595.948} C_VEL
LIN {X 0,Y 299.111,Z 998.362,A -85,B 0,C 180,E1 19601.876,E2 19601.876} C_VEL
LIN {X 0,Y 298.188,Z 986.502,A -85,B 0,C 180,E1 19608.322,E2 19608.322} C_VEL
LIN {X 0,Y 297.792,Z 980.007,A -85,B 0,C 180,E1 19614.184,E2 19614.184} C_VEL
LIN {X 0,Y 297.893,Z 977.905,A -85,B 0,C 180,E1 19620,E2 19620} C_VEL
LIN {X 0,Y 298.532,Z 980.849,A -85,B 0,C 180,E1 19625.802,E2 19625.802} C_VEL
LIN {X 0,Y 300.168,Z 989.058,A -85,B 0,C 180,E1 19632.337,E2 19632.337} C_VEL
LIN {X 0,Y 302.325,Z 1002.886,A -85,B 0,C 180,E1 19638.93,E2 19638.93} C_VEL
LIN {X 0,Y 302.795,Z 1013.871,A -85,B 0,C 180,E1 19642.628,E2 19642.628} C_VEL
LIN {X 0,Y 282.383,Z 1049.705,A -85,B 0,C 180,E1 19646.569,E2 19646.569} C_VEL
LIN {X 0,Y 260.128,Z 1082.232,A -85,B 0,C 180,E1 19652.015,E2 19652.015} C_VEL
LIN {X 0,Y 238.15,Z 1110.382,A -85,B 0,C 180,E1 19659.318,E2 19659.318} C_VEL
LIN {X 0,Y 219.455,Z 1132.962,A -85,B 0,C 180,E1 19668.522,E2 19668.522} C_VEL
LIN {X 0,Y 205.433,Z 1150.707,A -85,B 0,C 180,E1 19680.195,E2 19680.195} C_VEL
LIN {X 0,Y 198.786,Z 1161.631,A -85,B 0,C 180,E1 19692.324,E2 19692.324} C_VEL
LIN {X 0,Y 197.037,Z 1165.954,A -85,B 0,C 180,E1 19701.19,E2 19701.19} C_VEL
LIN {X 0,Y 197.228,Z 1167.417,A -85,B 0,C 180,E1 19710,E2 19710} C_VEL
LIN {X 0,Y 197.036,Z 1165.963,A -85,B 0,C 180,E1 19718.811,E2 19718.811} C_VEL
LIN {X 0,Y 199.263,Z 1160.462,A -85,B 0,C 180,E1 19729.313,E2 19729.313} C_VEL
LIN {X 0,Y 206.308,Z 1149.573,A -85,B 0,C 180,E1 19740.798,E2 19740.798} C_VEL
LIN {X 0,Y 220.591,Z 1131.616,A -85,B 0,C 180,E1 19752.181,E2 19752.181} C_VEL
LIN {X 0,Y 240.151,Z 1107.984,A -85,B 0,C 180,E1 19761.474,E2 19761.474} C_VEL
LIN {X 0,Y 262.214,Z 1079.456,A -85,B 0,C 180,E1 19768.581,E2 19768.581} C_VEL
LIN {X 0,Y 284.529,Z 1046.337,A -85,B 0,C 180,E1 19773.917,E2 19773.917} C_VEL
LIN {X 0,Y 302.838,Z 1014.071,A -85,B 0,C 180,E1 19777.364,E2 19777.364} C_VEL
LIN {X 0,Y 302.413,Z 1003.011,A -85,B 0,C 180,E1 19781.076,E2 19781.076} C_VEL
LIN {X 0,Y 300.282,Z 989.195,A -85,B 0,C 180,E1 19787.668,E2 19787.668} C_VEL
LIN {X 0,Y 298.619,Z 981.111,A -85,B 0,C 180,E1 19794.199,E2 19794.199} C_VEL
LIN {X 0,Y 298.312,Z 978.868,A -85,B 0,C 180,E1 19797.1,E2 19797.1} C_VEL
LIN {X 0,Y 297.898,Z 978.593,A -85,B 0,C 180,E1 19802.903,E2 19802.903} C_VEL
LIN {X 0,Y 297.909,Z 983.195,A -85,B 0,C 180,E1 19808.74,E2 19808.74} C_VEL
LIN {X 0,Y 298.77,Z 991.707,A -85,B 0,C 180,E1 19814.627,E2 19814.627} C_VEL
LIN {X 0,Y 299.585,Z 1004.637,A -85,B 0,C 180,E1 19820.645,E2 19820.645} C_VEL
LIN {X 0,Y 299.183,Z 1014.932,A -85,B 0,C 180,E1 19824.191,E2 19824.191} C_VEL
LIN {X 0,Y 292.357,Z 1026.918,A -85,B 0,C 180,E1 19825.516,E2 19825.516} C_VEL
LIN {X 0,Y 282.266,Z 1040.456,A -85,B 0,C 180,E1 19826.497,E2 19826.497} C_VEL
LIN {X 0,Y 273.004,Z 1051.787,A -85,B 0,C 180,E1 19827.445,E2 19827.445} C_VEL
LIN {X 0,Y 271.889,Z 1053.279,A -85,B 0,C 180,E1 19827.677,E2 19827.677} C_VEL
LIN {X 0,Y 249.237,Z 1082.908,A -85,B 0,C 180,E1 19833.643,E2 19833.643} C_VEL
LIN {X 0,Y 228.025,Z 1107.287,A -85,B 0,C 180,E1 19841.276,E2 19841.276} C_VEL
LIN {X 0,Y 209.901,Z 1126.794,A -85,B 0,C 180,E1 19850.972,E2 19850.972} C_VEL
LIN {X 0,Y 197.084,Z 1141.036,A -85,B 0,C 180,E1 19862.651,E2 19862.651} C_VEL
LIN {X 0,Y 191.109,Z 1148.895,A -85,B 0,C 180,E1 19873.956,E2 19873.956} C_VEL
LIN {X 0,Y 189.192,Z 1152.616,A -85,B 0,C 180,E1 19885.425,E2 19885.425} C_VEL
LIN {X 0,Y 189.375,Z 1152.919,A -85,B 0,C 180,E1 19890,E2 19890} C_VEL
LIN {X 0,Y 189.509,Z 1151.624,A -85,B 0,C 180,E1 19899.163,E2 19899.163} C_VEL
LIN {X 0,Y 192.702,Z 1146.564,A -85,B 0,C 180,E1 19910.007,E2 19910.007} C_VEL
LIN {X 0,Y 200.963,Z 1136.431,A -85,B 0,C 180,E1 19921.71,E2 19921.71} C_VEL
LIN {X 0,Y 216.637,Z 1119.516,A -85,B 0,C 180,E1 19933.078,E2 19933.078} C_VEL
LIN {X 0,Y 236.913,Z 1097.296,A -85,B 0,C 180,E1 19942.164,E2 19942.164} C_VEL
LIN {X 0,Y 259.645,Z 1069.777,A -85,B 0,C 180,E1 19949.216,E2 19949.216} C_VEL
LIN {X 0,Y 281.763,Z 1038.604,A -85,B 0,C 180,E1 19954.376,E2 19954.376} C_VEL
LIN {X 0,Y 294.314,Z 1017.378,A -85,B 0,C 180,E1 19957.027,E2 19957.027} C_VEL
LIN {X 0,Y 294.464,Z 1002.204,A -85,B 0,C 180,E1 19963.342,E2 19963.342} C_VEL
LIN {X 0,Y 294.032,Z 991.768,A -85,B 0,C 180,E1 19969.653,E2 19969.653} C_VEL
LIN {X 0,Y 293.884,Z 987.088,A -85,B 0,C 180,E1 19974.106,E2 19974.106} C_VEL
LIN {X 0,Y 294.19,Z 984.894,A -85,B 0,C 180,E1 19980,E2 19980} C_VEL
LIN {X 0,Y 294.687,Z 987.941,A -85,B 0,C 180,E1 19985.878,E2 19985.878} C_VEL
LIN {X 0,Y 296.176,Z 996.412,A -85,B 0,C 180,E1 19992.505,E2 19992.505} C_VEL
LIN {X 0,Y 297.647,Z 1009.298,A -85,B 0,C 180,E1 19998.686,E2 19998.686} C_VEL
LIN {X 0,Y 297.992,Z 1016.015,A -85,B 0,C 180,E1 20001.212,E2 20001.212} C_VEL
LIN {X 0,Y 294.924,Z 1022.626,A -85,B 0,C 180,E1 20002.037,E2 20002.037} C_VEL
LIN {X 0,Y 272.205,Z 1059.291,A -85,B 0,C 180,E1 20006.434,E2 20006.434} C_VEL
LIN {X 0,Y 249.693,Z 1089.915,A -85,B 0,C 180,E1 20012.212,E2 20012.212} C_VEL
LIN {X 0,Y 227.031,Z 1117.012,A -85,B 0,C 180,E1 20020.149,E2 20020.149} C_VEL
LIN {X 0,Y 207.96,Z 1138.892,A -85,B 0,C 180,E1 20030.586,E2 20030.586} C_VEL
LIN {X 0,Y 195.638,Z 1154.032,A -85,B 0,C 180,E1 20042.433,E2 20042.433} C_VEL
LIN {X 0,Y 190.406,Z 1162.603,A -85,B 0,C 180,E1 20053.896,E2 20053.896} C_VEL
LIN {X 0,Y 189.07,Z 1166.745,A -85,B 0,C 180,E1 20065.423,E2 20065.423} C_VEL
LIN {X 0,Y 189.33,Z 1167.121,A -85,B 0,C 180,E1 20070,E2 20070} C_VEL
LIN {X 0,Y 189.144,Z 1165.664,A -85,B 0,C 180,E1 20079.182,E2 20079.182} C_VEL
LIN {X 0,Y 191.775,Z 1159.889,A -85,B 0,C 180,E1 20090.497,E2 20090.497} C_VEL
LIN {X 0,Y 199.259,Z 1149.265,A -85,B 0,C 180,E1 20102.014,E2 20102.014} C_VEL
LIN {X 0,Y 213.512,Z 1132.474,A -85,B 0,C 180,E1 20113.079,E2 20113.079} C_VEL
LIN {X 0,Y 234.249,Z 1108.71,A -85,B 0,C 180,E1 20122.735,E2 20122.735} C_VEL
LIN {X 0,Y 257.698,Z 1079.592,A -85,B 0,C 180,E1 20130.055,E2 20130.055} C_VEL
LIN {X 0,Y 280.598,Z 1046.771,A -85,B 0,C 180,E1 20135.314,E2 20135.314} C_VEL
LIN {X 0,Y 297.578,Z 1017.954,A -85,B 0,C 180,E1 20138.405,E2 20138.405} C_VEL
LIN {X 0,Y 297.879,Z 1010.884,A -85,B 0,C 180,E1 20140.742,E2 20140.742} C_VEL
LIN {X 0,Y 296.3,Z 996.529,A -85,B 0,C 180,E1 20147.5,E2 20147.5} C_VEL
LIN {X 0,Y 294.776,Z 988.173,A -85,B 0,C 180,E1 20154.124,E2 20154.124} C_VEL
LIN {X 0,Y 294.58,Z 985.879,A -85,B 0,C 180,E1 20157.064,E2 20157.064} C_VEL
LIN {X 0,Y 294.114,Z 985.607,A -85,B 0,C 180,E1 20162.941,E2 20162.941} C_VEL
LIN {X 0,Y 293.989,Z 990.339,A -85,B 0,C 180,E1 20168.857,E2 20168.857} C_VEL
LIN {X 0,Y 294.419,Z 999.014,A -85,B 0,C 180,E1 20174.848,E2 20174.848} C_VEL
LIN {X 0,Y 294.683,Z 1012.342,A -85,B 0,C 180,E1 20181.004,E2 20181.004} C_VEL
LIN {X 0,Y 294.391,Z 1017.965,A -85,B 0,C 180,E1 20183.066,E2 20183.066} C_VEL
LIN {X 0,Y 273.681,Z 1050.791,A -85,B 0,C 180,E1 20187.269,E2 20187.269} C_VEL
LIN {X 0,Y 271.889,Z 1053.279,A -85,B 0,C 180,E1 20187.677,E2 20187.677} C_VEL
LIN {X 0,Y 261.048,Z 1065.576,A -85,B 0,C 180,E1 20189.058,E2 20189.058} C_VEL
LIN {X 0,Y 249.949,Z 1077.12,A -85,B 0,C 180,E1 20190.626,E2 20190.626} C_VEL
LIN {X 0,Y 228.332,Z 1101.663,A -85,B 0,C 180,E1 20197.527,E2 20197.527} C_VEL
LIN {X 0,Y 208.581,Z 1122.027,A -85,B 0,C 180,E1 20206.488,E2 20206.488} C_VEL
LIN {X 0,Y 194.007,Z 1136.872,A -85,B 0,C 180,E1 20217.011,E2 20217.011} C_VEL
LIN {X 0,Y 185.124,Z 1146.951,A -85,B 0,C 180,E1 20229.144,E2 20229.144} C_VEL
LIN {X 0,Y 181.649,Z 1151.956,A -85,B 0,C 180,E1 20240.436,E2 20240.436} C_VEL
LIN {X 0,Y 181.471,Z 1153.215,A -85,B 0,C 180,E1 20250,E2 20250} C_VEL
LIN {X 0,Y 181.662,Z 1151.922,A -85,B 0,C 180,E1 20259.563,E2 20259.563} C_VEL
LIN {X 0,Y 185.137,Z 1146.868,A -85,B 0,C 180,E1 20270.862,E2 20270.862} C_VEL
LIN {X 0,Y 194.081,Z 1136.738,A -85,B 0,C 180,E1 20282.974,E2 20282.974} C_VEL
LIN {X 0,Y 210.554,Z 1120.045,A -85,B 0,C 180,E1 20294.478,E2 20294.478} C_VEL
LIN {X 0,Y 232.432,Z 1097.096,A -85,B 0,C 180,E1 20303.918,E2 20303.918} C_VEL
LIN {X 0,Y 255.258,Z 1070.525,A -85,B 0,C 180,E1 20310.689,E2 20310.689} C_VEL
LIN {X 0,Y 278.693,Z 1038.401,A -85,B 0,C 180,E1 20315.938,E2 20315.938} C_VEL
LIN {X 0,Y 289.177,Z 1021.026,A -85,B 0,C 180,E1 20318.175,E2 20318.175} C_VEL
LIN {X 0,Y 289.794,Z 1007.495,A -85,B 0,C 180,E1 20324.136,E2 20324.136} C_VEL
LIN {X 0,Y 289.812,Z 998.78,A -85,B 0,C 180,E1 20329.5,E2 20329.5} C_VEL
LIN {X 0,Y 289.925,Z 994.142,A -85,B 0,C 180,E1 20334.025,E2 20334.025} C_VEL
LIN {X 0,Y 290.348,Z 991.81,A -85,B 0,C 180,E1 20340,E2 20340} C_VEL
LIN {X 0,Y 290.79,Z 994.993,A -85,B 0,C 180,E1 20345.957,E2 20345.957} C_VEL
LIN {X 0,Y 291.843,Z 1003.644,A -85,B 0,C 180,E1 20352.694,E2 20352.694} C_VEL
LIN {X 0,Y 292.775,Z 1016.102,A -85,B 0,C 180,E1 20358.664,E2 20358.664} C_VEL
LIN {X 0,Y 292.893,Z 1020.59,A -85,B 0,C 180,E1 20360.39,E2 20360.39} C_VEL
LIN {X 0,Y 271.21,Z 1055.262,A -85,B 0,C 180,E1 20364.361,E2 20364.361} C_VEL
LIN {X 0,Y 248.238,Z 1085.98,A -85,B 0,C 180,E1 20369.771,E2 20369.771} C_VEL
LIN {X 0,Y 226.155,Z 1111.81,A -85,B 0,C 180,E1 20376.804,E2 20376.804} C_VEL
LIN {X 0,Y 206.433,Z 1133.283,A -85,B 0,C 180,E1 20386.02,E2 20386.02} C_VEL
LIN {X 0,Y 191.234,Z 1150.166,A -85,B 0,C 180,E1 20397.817,E2 20397.817} C_VEL
LIN {X 0,Y 183.404,Z 1161.022,A -85,B 0,C 180,E1 20410.786,E2 20410.786} C_VEL
LIN {X 0,Y 181.29,Z 1165.356,A -85,B 0,C 180,E1 20420.418,E2 20420.418} C_VEL
LIN {X 0,Y 181.423,Z 1166.824,A -85,B 0,C 180,E1 20430,E2 20430} C_VEL
LIN {X 0,Y 181.285,Z 1165.365,A -85,B 0,C 180,E1 20439.584,E2 20439.584} C_VEL
LIN {X 0,Y 184.295,Z 1159.422,A -85,B 0,C 180,E1 20451.621,E2 20451.621} C_VEL
LIN {X 0,Y 192.343,Z 1148.958,A -85,B 0,C 180,E1 20463.311,E2 20463.311} C_VEL
LIN {X 0,Y 208.124,Z 1131.522,A -85,B 0,C 180,E1 20474.985,E2 20474.985} C_VEL
LIN {X 0,Y 229.537,Z 1108.177,A -85,B 0,C 180,E1 20484.445,E2 20484.445} C_VEL
LIN {X 0,Y 253.209,Z 1079.962,A -85,B 0,C 180,E1 20491.527,E2 20491.527} C_VEL
LIN {X 0,Y 277.447,Z 1046.25,A -85,B 0,C 180,E1 20496.864,E2 20496.864} C_VEL
LIN {X 0,Y 292.726,Z 1021.27,A -85,B 0,C 180,E1 20499.537,E2 20499.537} C_VEL
LIN {X 0,Y 292.519,Z 1009.588,A -85,B 0,C 180,E1 20504.287,E2 20504.287} C_VEL
LIN {X 0,Y 291.539,Z 1000.292,A -85,B 0,C 180,E1 20509.562,E2 20509.562} C_VEL
LIN {X 0,Y 290.722,Z 992.835,A -85,B 0,C 180,E1 20517.025,E2 20517.025} C_VEL
LIN {X 0,Y 290.493,Z 991.987,A -85,B 0,C 180,E1 20520,E2 20520} C_VEL
LIN {X 0,Y 290.019,Z 994.423,A -85,B 0,C 180,E1 20525.973,E2 20525.973} C_VEL
LIN {X 0,Y 289.936,Z 1001.2,A -85,B 0,C 180,E1 20532.015,E2 20532.015} C_VEL
LIN {X 0,Y 289.833,Z 1013.716,A -85,B 0,C 180,E1 20538.73,E2 20538.73} C_VEL
LIN {X 0,Y 288.818,Z 1022.491,A -85,B 0,C 180,E1 20542.07,E2 20542.07} C_VEL
LIN {X 0,Y 267.866,Z 1054.074,A -85,B 0,C 180,E1 20546.229,E2 20546.229} C_VEL
LIN {X 0,Y 249.949,Z 1077.12,A -85,B 0,C 180,E1 20550.626,E2 20550.626} C_VEL
LIN {X 0,Y 238.516,Z 1088.063,A -85,B 0,C 180,E1 20552.443,E2 20552.443} C_VEL
LIN {X 0,Y 227.132,Z 1098.178,A -85,B 0,C 180,E1 20554.548,E2 20554.548} C_VEL
LIN {X 0,Y 204.875,Z 1120.363,A -85,B 0,C 180,E1 20563.803,E2 20563.803} C_VEL
LIN {X 0,Y 187.226,Z 1137.176,A -85,B 0,C 180,E1 20575.653,E2 20575.653} C_VEL
LIN {X 0,Y 176.88,Z 1148.201,A -85,B 0,C 180,E1 20589.783,E2 20589.783} C_VEL
LIN {X 0,Y 173.797,Z 1152.255,A -85,B 0,C 180,E1 20599.999,E2 20599.999} C_VEL
LIN {X 0,Y 173.578,Z 1153.511,A -85,B 0,C 180,E1 20609.999,E2 20609.999} C_VEL
LIN {X 0,Y 173.81,Z 1152.221,A -85,B 0,C 180,E1 20619.999,E2 20619.999} C_VEL
LIN {X 0,Y 177.939,Z 1146.782,A -85,B 0,C 180,E1 20632.431,E2 20632.431} C_VEL
LIN {X 0,Y 188.447,Z 1135.911,A -85,B 0,C 180,E1 20645.314,E2 20645.314} C_VEL
LIN {X 0,Y 205.109,Z 1120.045,A -85,B 0,C 180,E1 20656.239,E2 20656.239} C_VEL
LIN {X 0,Y 227.5,Z 1097.65,A -85,B 0,C 180,E1 20665.5,E2 20665.5} C_VEL
LIN {X 0,Y 251.39,Z 1070.835,A -85,B 0,C 180,E1 20672.298,E2 20672.298} C_VEL
LIN {X 0,Y 275.368,Z 1038.913,A -85,B 0,C 180,E1 20677.444,E2 20677.444} C_VEL
LIN {X 0,Y 283.859,Z 1025.856,A -85,B 0,C 180,E1 20678.995,E2 20678.995} C_VEL
LIN {X 0,Y 285.081,Z 1013.28,A -85,B 0,C 180,E1 20684.654,E2 20684.654} C_VEL
LIN {X 0,Y 285.509,Z 1004.035,A -85,B 0,C 180,E1 20690.877,E2 20690.877} C_VEL
LIN {X 0,Y 286.015,Z 999.151,A -85,B 0,C 180,E1 20696.976,E2 20696.976} C_VEL
LIN {X 0,Y 286.313,Z 998.598,A -85,B 0,C 180,E1 20700,E2 20700} C_VEL
LIN {X 0,Y 286.593,Z 1001.879,A -85,B 0,C 180,E1 20706.045,E2 20706.045} C_VEL
LIN {X 0,Y 287.367,Z 1009.567,A -85,B 0,C 180,E1 20712.125,E2 20712.125} C_VEL
LIN {X 0,Y 287.824,Z 1022.102,A -85,B 0,C 180,E1 20718.334,E2 20718.334} C_VEL
LIN {X 0,Y 287.78,Z 1024.491,A -85,B 0,C 180,E1 20719.291,E2 20719.291} C_VEL
LIN {X 0,Y 264.891,Z 1059.316,A -85,B 0,C 180,E1 20723.383,E2 20723.383} C_VEL
LIN {X 0,Y 240.144,Z 1090.64,A -85,B 0,C 180,E1 20729.199,E2 20729.199} C_VEL
LIN {X 0,Y 216.157,Z 1117.002,A -85,B 0,C 180,E1 20737.041,E2 20737.041} C_VEL
LIN {X 0,Y 195.388,Z 1138.311,A -85,B 0,C 180,E1 20747.527,E2 20747.527} C_VEL
LIN {X 0,Y 181.252,Z 1153.415,A -85,B 0,C 180,E1 20760.032,E2 20760.032} C_VEL
LIN {X 0,Y 175.331,Z 1161.382,A -85,B 0,C 180,E1 20771.209,E2 20771.209} C_VEL
LIN {X 0,Y 173.41,Z 1165.056,A -85,B 0,C 180,E1 20779.978,E2 20779.978} C_VEL
LIN {X 0,Y 173.528,Z 1166.528,A -85,B 0,C 180,E1 20790.001,E2 20790.001} C_VEL
LIN {X 0,Y 173.402,Z 1165.066,A -85,B 0,C 180,E1 20800.024,E2 20800.024} C_VEL
LIN {X 0,Y 176.758,Z 1159.118,A -85,B 0,C 180,E1 20812.593,E2 20812.593} C_VEL
LIN {X 0,Y 185.497,Z 1148.649,A -85,B 0,C 180,E1 20824.712,E2 20824.712} C_VEL
LIN {X 0,Y 202.35,Z 1131.211,A -85,B 0,C 180,E1 20836.645,E2 20836.645} C_VEL
LIN {X 0,Y 224.866,Z 1107.872,A -85,B 0,C 180,E1 20846.146,E2 20846.146} C_VEL
LIN {X 0,Y 249.412,Z 1079.658,A -85,B 0,C 180,E1 20853.179,E2 20853.179} C_VEL
LIN {X 0,Y 273.823,Z 1046.778,A -85,B 0,C 180,E1 20858.324,E2 20858.324} C_VEL
LIN {X 0,Y 287.818,Z 1024.724,A -85,B 0,C 180,E1 20860.689,E2 20860.689} C_VEL
LIN {X 0,Y 287.61,Z 1012.319,A -85,B 0,C 180,E1 20866.344,E2 20866.344} C_VEL
LIN {X 0,Y 286.816,Z 1003.615,A -85,B 0,C 180,E1 20872.442,E2 20872.442} C_VEL
LIN {X 0,Y 286.633,Z 999.678,A -85,B 0,C 180,E1 20876.982,E2 20876.982} C_VEL
LIN {X 0,Y 286.445,Z 998.781,A -85,B 0,C 180,E1 20880,E2 20880} C_VEL
LIN {X 0,Y 285.793,Z 1001.32,A -85,B 0,C 180,E1 20886.061,E2 20886.061} C_VEL
LIN {X 0,Y 285.379,Z 1009.498,A -85,B 0,C 180,E1 20892.986,E2 20892.986} C_VEL
LIN {X 0,Y 284.682,Z 1021.215,A -85,B 0,C 180,E1 20899.082,E2 20899.082} C_VEL
LIN {X 0,Y 283.739,Z 1026.31,A -85,B 0,C 180,E1 20900.944,E2 20900.944} C_VEL
LIN {X 0,Y 260.951,Z 1058.943,A -85,B 0,C 180,E1 20905.405,E2 20905.405} C_VEL
LIN {X 0,Y 236.644,Z 1087.932,A -85,B 0,C 180,E1 20911.553,E2 20911.553} C_VEL
LIN {X 0,Y 227.132,Z 1098.178,A -85,B 0,C 180,E1 20914.548,E2 20914.548} C_VEL
LIN {X 0,Y 215.65,Z 1107.639,A -85,B 0,C 180,E1 20916.968,E2 20916.968} C_VEL
LIN {X 0,Y 205.31,Z 1115.147,A -85,B 0,C 180,E1 20919.314,E2 20919.314} C_VEL
LIN {X 0,Y 204.196,Z 1116.102,A -85,B 0,C 180,E1 20919.769,E2 20919.769} C_VEL
LIN {X 0,Y 184.924,Z 1133.537,A -85,B 0,C 180,E1 20930.691,E2 20930.691} C_VEL
LIN {X 0,Y 172.015,Z 1145.657,A -85,B 0,C 180,E1 20943.983,E2 20943.983} C_VEL
LIN {X 0,Y 167.229,Z 1150.934,A -85,B 0,C 180,E1 20954.293,E2 20954.293} C_VEL
LIN {X 0,Y 165.509,Z 1153.507,A -85,B 0,C 180,E1 20964.768,E2 20964.768} C_VEL
LIN {X 0,Y 165.699,Z 1153.807,A -85,B 0,C 180,E1 20969.999,E2 20969.999} C_VEL
LIN {X 0,Y 165.996,Z 1152.519,A -85,B 0,C 180,E1 20980.475,E2 20980.475} C_VEL
LIN {X 0,Y 170.496,Z 1147.084,A -85,B 0,C 180,E1 20993.47,E2 20993.47} C_VEL
LIN {X 0,Y 181.752,Z 1136.318,A -85,B 0,C 180,E1 21006.708,E2 21006.708} C_VEL
LIN {X 0,Y 199.612,Z 1120.306,A -85,B 0,C 180,E1 21017.951,E2 21017.951} C_VEL
LIN {X 0,Y 223.043,Z 1097.913,A -85,B 0,C 180,E1 21027.233,E2 21027.233} C_VEL
LIN {X 0,Y 247.732,Z 1071.139,A -85,B 0,C 180,E1 21033.957,E2 21033.957} C_VEL
LIN {X 0,Y 271.806,Z 1040.065,A -85,B 0,C 180,E1 21038.9,E2 21038.9} C_VEL
LIN {X 0,Y 279.047,Z 1029.215,A -85,B 0,C 180,E1 21040.247,E2 21040.247} C_VEL
LIN {X 0,Y 280.397,Z 1018.231,A -85,B 0,C 180,E1 21045.627,E2 21045.627} C_VEL
LIN {X 0,Y 281.008,Z 1010.871,A -85,B 0,C 180,E1 21050.73,E2 21050.73} C_VEL
LIN {X 0,Y 281.84,Z 1005.934,A -85,B 0,C 180,E1 21056.931,E2 21056.931} C_VEL
LIN {X 0,Y 282.166,Z 1005.326,A -85,B 0,C 180,E1 21060,E2 21060} C_VEL
LIN {X 0,Y 282.31,Z 1007.43,A -85,B 0,C 180,E1 21064.599,E2 21064.599} C_VEL
LIN {X 0,Y 282.669,Z 1015.324,A -85,B 0,C 180,E1 21071.548,E2 21071.548} C_VEL
LIN {X 0,Y 282.672,Z 1027.651,A -85,B 0,C 180,E1 21077.88,E2 21077.88} C_VEL
LIN {X 0,Y 279.147,Z 1033.902,A -85,B 0,C 180,E1 21078.696,E2 21078.696} C_VEL
LIN {X 0,Y 253.992,Z 1069.115,A -85,B 0,C 180,E1 21083.293,E2 21083.293} C_VEL
LIN {X 0,Y 227.816,Z 1099.575,A -85,B 0,C 180,E1 21089.753,E2 21089.753} C_VEL
LIN {X 0,Y 203.269,Z 1124.618,A -85,B 0,C 180,E1 21098.571,E2 21098.571} C_VEL
LIN {X 0,Y 184.484,Z 1142.677,A -85,B 0,C 180,E1 21109.129,E2 21109.129} C_VEL
LIN {X 0,Y 171.481,Z 1156.11,A -85,B 0,C 180,E1 21122.44,E2 21122.44} C_VEL
LIN {X 0,Y 166.513,Z 1162.947,A -85,B 0,C 180,E1 21134.225,E2 21134.225} C_VEL
LIN {X 0,Y 165.32,Z 1165.851,A -85,B 0,C 180,E1 21144.763,E2 21144.763} C_VEL
LIN {X 0,Y 165.631,Z 1166.232,A -85,B 0,C 180,E1 21150.001,E2 21150.001} C_VEL
LIN {X 0,Y 165.553,Z 1164.767,A -85,B 0,C 180,E1 21160.504,E2 21160.504} C_VEL
LIN {X 0,Y 169.274,Z 1158.813,A -85,B 0,C 180,E1 21173.651,E2 21173.651} C_VEL
LIN {X 0,Y 178.783,Z 1148.341,A -85,B 0,C 180,E1 21186.217,E2 21186.217} C_VEL
LIN {X 0,Y 196.776,Z 1130.903,A -85,B 0,C 180,E1 21198.392,E2 21198.392} C_VEL
LIN {X 0,Y 220.351,Z 1107.563,A -85,B 0,C 180,E1 21207.938,E2 21207.938} C_VEL
LIN {X 0,Y 245.938,Z 1079.212,A -85,B 0,C 180,E1 21214.909,E2 21214.909} C_VEL
LIN {X 0,Y 271.078,Z 1046.245,A -85,B 0,C 180,E1 21219.949,E2 21219.949} C_VEL
LIN {X 0,Y 282.133,Z 1029.378,A -85,B 0,C 180,E1 21221.755,E2 21221.755} C_VEL
LIN {X 0,Y 282.913,Z 1024.13,A -85,B 0,C 180,E1 21223.76,E2 21223.76} C_VEL
LIN {X 0,Y 282.772,Z 1014.236,A -85,B 0,C 180,E1 21229.235,E2 21229.235} C_VEL
LIN {X 0,Y 282.443,Z 1006.489,A -85,B 0,C 180,E1 21236.937,E2 21236.937} C_VEL
LIN {X 0,Y 282.308,Z 1005.496,A -85,B 0,C 180,E1 21240,E2 21240} C_VEL
LIN {X 0,Y 281.472,Z 1008.152,A -85,B 0,C 180,E1 21246.155,E2 21246.155} C_VEL
LIN {X 0,Y 280.788,Z 1015.304,A -85,B 0,C 180,E1 21252.413,E2 21252.413} C_VEL
LIN {X 0,Y 279.627,Z 1026.409,A -85,B 0,C 180,E1 21258.435,E2 21258.435} C_VEL
LIN {X 0,Y 278.987,Z 1029.676,A -85,B 0,C 180,E1 21259.755,E2 21259.755} C_VEL
LIN {X 0,Y 254.913,Z 1062.623,A -85,B 0,C 180,E1 21264.343,E2 21264.343} C_VEL
LIN {X 0,Y 229.867,Z 1091.093,A -85,B 0,C 180,E1 21270.62,E2 21270.62} C_VEL
LIN {X 0,Y 205.855,Z 1114.617,A -85,B 0,C 180,E1 21279.035,E2 21279.035} C_VEL
LIN {X 0,Y 204.196,Z 1116.102,A -85,B 0,C 180,E1 21279.769,E2 21279.769} C_VEL
LIN {X 0,Y 193.038,Z 1123.861,A -85,B 0,C 180,E1 21282.987,E2 21282.987} C_VEL
LIN {X 0,Y 182.256,Z 1130.788,A -85,B 0,C 180,E1 21286.641,E2 21286.641} C_VEL
LIN {X 0,Y 167.609,Z 1143.314,A -85,B 0,C 180,E1 21299.013,E2 21299.013} C_VEL
LIN {X 0,Y 159.528,Z 1151.234,A -85,B 0,C 180,E1 21313.514,E2 21313.514} C_VEL
LIN {X 0,Y 157.608,Z 1153.804,A -85,B 0,C 180,E1 21324.505,E2 21324.505} C_VEL
LIN {X 0,Y 157.793,Z 1154.103,A -85,B 0,C 180,E1 21329.999,E2 21329.999} C_VEL
LIN {X 0,Y 158.162,Z 1152.818,A -85,B 0,C 180,E1 21341,E2 21341} C_VEL
LIN {X 0,Y 163.121,Z 1147.388,A -85,B 0,C 180,E1 21354.6,E2 21354.6} C_VEL
LIN {X 0,Y 174.136,Z 1137.655,A -85,B 0,C 180,E1 21367.343,E2 21367.343} C_VEL
LIN {X 0,Y 194.427,Z 1120.461,A -85,B 0,C 180,E1 21379.812,E2 21379.812} C_VEL
LIN {X 0,Y 218.75,Z 1098.22,A -85,B 0,C 180,E1 21389.024,E2 21389.024} C_VEL
LIN {X 0,Y 244.283,Z 1071.445,A -85,B 0,C 180,E1 21395.665,E2 21395.665} C_VEL
LIN {X 0,Y 270.069,Z 1038.859,A -85,B 0,C 180,E1 21400.678,E2 21400.678} C_VEL
LIN {X 0,Y 274.037,Z 1032.747,A -85,B 0,C 180,E1 21401.558,E2 21401.558} C_VEL
LIN {X 0,Y 275.775,Z 1021.964,A -85,B 0,C 180,E1 21407.358,E2 21407.358} C_VEL
LIN {X 0,Y 276.869,Z 1014.558,A -85,B 0,C 180,E1 21413.743,E2 21413.743} C_VEL
LIN {X 0,Y 277.806,Z 1011.906,A -85,B 0,C 180,E1 21420,E2 21420} C_VEL
LIN {X 0,Y 277.828,Z 1014.093,A -85,B 0,C 180,E1 21424.673,E2 21424.673} C_VEL
LIN {X 0,Y 278.002,Z 1021.071,A -85,B 0,C 180,E1 21430.953,E2 21430.953} C_VEL
LIN {X 0,Y 277.64,Z 1031.101,A -85,B 0,C 180,E1 21436.497,E2 21436.497} C_VEL
LIN {X 0,Y 276.421,Z 1033.962,A -85,B 0,C 180,E1 21437.141,E2 21437.141} C_VEL
LIN {X 0,Y 251.092,Z 1068.507,A -85,B 0,C 180,E1 21441.524,E2 21441.524} C_VEL
LIN {X 0,Y 224.044,Z 1099.066,A -85,B 0,C 180,E1 21447.87,E2 21447.87} C_VEL
LIN {X 0,Y 198.016,Z 1124.467,A -85,B 0,C 180,E1 21456.772,E2 21456.772} C_VEL
LIN {X 0,Y 176.682,Z 1143.854,A -85,B 0,C 180,E1 21468.556,E2 21468.556} C_VEL
LIN {X 0,Y 163.355,Z 1156.83,A -85,B 0,C 180,E1 21482.492,E2 21482.492} C_VEL
LIN {X 0,Y 158.764,Z 1162.644,A -85,B 0,C 180,E1 21493.433,E2 21493.433} C_VEL
LIN {X 0,Y 157.401,Z 1165.553,A -85,B 0,C 180,E1 21504.499,E2 21504.499} C_VEL
LIN {X 0,Y 157.72,Z 1165.936,A -85,B 0,C 180,E1 21510.001,E2 21510.001} C_VEL
LIN {X 0,Y 157.682,Z 1164.466,A -85,B 0,C 180,E1 21521.035,E2 21521.035} C_VEL
LIN {X 0,Y 161.83,Z 1158.507,A -85,B 0,C 180,E1 21534.811,E2 21534.811} C_VEL
LIN {X 0,Y 173.472,Z 1146.795,A -85,B 0,C 180,E1 21548.938,E2 21548.938} C_VEL
LIN {X 0,Y 191.378,Z 1130.594,A -85,B 0,C 180,E1 21560.246,E2 21560.246} C_VEL
LIN {X 0,Y 215.85,Z 1107.447,A -85,B 0,C 180,E1 21569.755,E2 21569.755} C_VEL
LIN {X 0,Y 242.486,Z 1079.026,A -85,B 0,C 180,E1 21576.638,E2 21576.638} C_VEL
LIN {X 0,Y 268.4,Z 1045.944,A -85,B 0,C 180,E1 21581.579,E2 21581.579} C_VEL
LIN {X 0,Y 277.359,Z 1032.763,A -85,B 0,C 180,E1 21582.983,E2 21582.983} C_VEL
LIN {X 0,Y 278.135,Z 1022.491,A -85,B 0,C 180,E1 21588.181,E2 21588.181} C_VEL
LIN {X 0,Y 277.921,Z 1014.293,A -85,B 0,C 180,E1 21595.328,E2 21595.328} C_VEL
LIN {X 0,Y 277.928,Z 1012.091,A -85,B 0,C 180,E1 21600,E2 21600} C_VEL
LIN {X 0,Y 276.935,Z 1014.859,A -85,B 0,C 180,E1 21606.256,E2 21606.256} C_VEL
LIN {X 0,Y 275.854,Z 1022.248,A -85,B 0,C 180,E1 21612.639,E2 21612.639} C_VEL
LIN {X 0,Y 274.252,Z 1032.781,A -85,B 0,C 180,E1 21618.385,E2 21618.385} C_VEL
LIN {X 0,Y 250.473,Z 1064.331,A -85,B 0,C 180,E1 21622.915,E2 21622.915} C_VEL
LIN {X 0,Y 224.66,Z 1092.525,A -85,B 0,C 180,E1 21629.167,E2 21629.167} C_VEL
LIN {X 0,Y 200.614,Z 1115.098,A -85,B 0,C 180,E1 21637.314,E2 21637.314} C_VEL
LIN {X 0,Y 182.256,Z 1130.788,A -85,B 0,C 180,E1 21646.641,E2 21646.641} C_VEL
LIN {X 0,Y 172.046,Z 1136.888,A -85,B 0,C 180,E1 21650.82,E2 21650.82} C_VEL
LIN {X 0,Y 162.545,Z 1142.141,A -85,B 0,C 180,E1 21655.546,E2 21655.546} C_VEL
LIN {X 0,Y 153.248,Z 1150.102,A -85,B 0,C 180,E1 21669.064,E2 21669.064} C_VEL
LIN {X 0,Y 149.724,Z 1154.101,A -85,B 0,C 180,E1 21684.215,E2 21684.215} C_VEL
LIN {X 0,Y 149.908,Z 1154.399,A -85,B 0,C 180,E1 21689.999,E2 21689.999} C_VEL
LIN {X 0,Y 150.34,Z 1153.118,A -85,B 0,C 180,E1 21701.58,E2 21701.58} C_VEL
LIN {X 0,Y 155.817,Z 1147.691,A -85,B 0,C 180,E1 21715.836,E2 21715.836} C_VEL
LIN {X 0,Y 167.731,Z 1137.962,A -85,B 0,C 180,E1 21729.032,E2 21729.032} C_VEL
LIN {X 0,Y 188.501,Z 1121.42,A -85,B 0,C 180,E1 21741.359,E2 21741.359} C_VEL
LIN {X 0,Y 214.787,Z 1098.421,A -85,B 0,C 180,E1 21750.918,E2 21750.918} C_VEL
LIN {X 0,Y 241.058,Z 1071.752,A -85,B 0,C 180,E1 21757.419,E2 21757.419} C_VEL
LIN {X 0,Y 267.515,Z 1039.163,A -85,B 0,C 180,E1 21762.305,E2 21762.305} C_VEL
LIN {X 0,Y 268.916,Z 1037.152,A -85,B 0,C 180,E1 21762.543,E2 21762.543} C_VEL
LIN {X 0,Y 271.008,Z 1027.232,A -85,B 0,C 180,E1 21768.206,E2 21768.206} C_VEL
LIN {X 0,Y 272.193,Z 1021.208,A -85,B 0,C 180,E1 21773.635,E2 21773.635} C_VEL
LIN {X 0,Y 272.866,Z 1019.188,A -85,B 0,C 180,E1 21776.83,E2 21776.83} C_VEL
LIN {X 0,Y 273.363,Z 1018.435,A -85,B 0,C 180,E1 21780,E2 21780} C_VEL
LIN {X 0,Y 273.31,Z 1020.731,A -85,B 0,C 180,E1 21784.752,E2 21784.752} C_VEL
LIN {X 0,Y 273.047,Z 1027.87,A -85,B 0,C 180,E1 21791.154,E2 21791.154} C_VEL
LIN {X 0,Y 272.531,Z 1035.849,A -85,B 0,C 180,E1 21795.66,E2 21795.66} C_VEL
LIN {X 0,Y 246.475,Z 1070.234,A -85,B 0,C 180,E1 21800.098,E2 21800.098} C_VEL
LIN {X 0,Y 218.911,Z 1100.105,A -85,B 0,C 180,E1 21806.347,E2 21806.347} C_VEL
LIN {X 0,Y 193.034,Z 1124.243,A -85,B 0,C 180,E1 21814.834,E2 21814.834} C_VEL
LIN {X 0,Y 170.595,Z 1143.543,A -85,B 0,C 180,E1 21826.723,E2 21826.723} C_VEL
LIN {X 0,Y 156.147,Z 1156.523,A -85,B 0,C 180,E1 21841.106,E2 21841.106} C_VEL
LIN {X 0,Y 151.076,Z 1162.343,A -85,B 0,C 180,E1 21852.564,E2 21852.564} C_VEL
LIN {X 0,Y 149.491,Z 1165.255,A -85,B 0,C 180,E1 21864.207,E2 21864.207} C_VEL
LIN {X 0,Y 149.807,Z 1165.639,A -85,B 0,C 180,E1 21870.001,E2 21870.001} C_VEL
LIN {X 0,Y 149.821,Z 1164.166,A -85,B 0,C 180,E1 21881.622,E2 21881.622} C_VEL
LIN {X 0,Y 154.452,Z 1158.202,A -85,B 0,C 180,E1 21896.083,E2 21896.083} C_VEL
LIN {X 0,Y 165.757,Z 1147.724,A -85,B 0,C 180,E1 21909.589,E2 21909.589} C_VEL
LIN {X 0,Y 186.189,Z 1130.285,A -85,B 0,C 180,E1 21922.206,E2 21922.206} C_VEL
LIN {X 0,Y 212.696,Z 1106.274,A -85,B 0,C 180,E1 21931.934,E2 21931.934} C_VEL
LIN {X 0,Y 239.842,Z 1078.149,A -85,B 0,C 180,E1 21938.54,E2 21938.54} C_VEL
LIN {X 0,Y 265.951,Z 1045.644,A -85,B 0,C 180,E1 21943.235,E2 21943.235} C_VEL
LIN {X 0,Y 272.617,Z 1035.97,A -85,B 0,C 180,E1 21944.345,E2 21944.345} C_VEL
LIN {X 0,Y 273.245,Z 1025.756,A -85,B 0,C 180,E1 21950.464,E2 21950.464} C_VEL
LIN {X 0,Y 273.5,Z 1019.767,A -85,B 0,C 180,E1 21956.837,E2 21956.837} C_VEL
LIN {X 0,Y 273.488,Z 1018.615,A -85,B 0,C 180,E1 21960,E2 21960} C_VEL
LIN {X 0,Y 272.56,Z 1020.369,A -85,B 0,C 180,E1 21964.749,E2 21964.749} C_VEL
LIN {X 0,Y 271.373,Z 1026.05,A -85,B 0,C 180,E1 21970.773,E2 21970.773} C_VEL
LIN {X 0,Y 269.351,Z 1036.295,A -85,B 0,C 180,E1 21976.985,E2 21976.985} C_VEL
LIN {X 0,Y 267.149,Z 1039.909,A -85,B 0,C 180,E1 21977.66,E2 21977.66} C_VEL
LIN {X 0,Y 240.959,Z 1072.049,A -85,B 0,C 180,E1 21982.522,E2 21982.522} C_VEL
LIN {X 0,Y 213.143,Z 1100.115,A -85,B 0,C 180,E1 21989.492,E2 21989.492} C_VEL
LIN {X 0,Y 188.102,Z 1121.828,A -85,B 0,C 180,E1 21998.723,E2 21998.723} C_VEL
LIN {X 0,Y 167.635,Z 1138.088,A -85,B 0,C 180,E1 22010.94,E2 22010.94} C_VEL
LIN {X 0,Y 162.545,Z 1142.141,A -85,B 0,C 180,E1 22015.546,E2 22015.546} C_VEL
LIN {X 0,Y 153.996,Z 1146.588,A -85,B 0,C 180,E1 22020.846,E2 22020.846} C_VEL
LIN {X 0,Y 146.307,Z 1149.951,A -85,B 0,C 180,E1 22026.765,E2 22026.765} C_VEL
LIN {X 0,Y 142.519,Z 1153.449,A -85,B 0,C 180,E1 22037.774,E2 22037.774} C_VEL
LIN {X 0,Y 142,Z 1154.696,A -85,B 0,C 180,E1 22049.999,E2 22049.999} C_VEL
LIN {X 0,Y 142.533,Z 1153.417,A -85,B 0,C 180,E1 22062.224,E2 22062.224} C_VEL
LIN {X 0,Y 148.583,Z 1147.995,A -85,B 0,C 180,E1 22077.194,E2 22077.194} C_VEL
LIN {X 0,Y 161.494,Z 1138.268,A -85,B 0,C 180,E1 22090.85,E2 22090.85} C_VEL
LIN {X 0,Y 183.436,Z 1121.782,A -85,B 0,C 180,E1 22103.328,E2 22103.328} C_VEL
LIN {X 0,Y 209.946,Z 1099.676,A -85,B 0,C 180,E1 22112.562,E2 22112.562} C_VEL
LIN {X 0,Y 238.064,Z 1072.059,A -85,B 0,C 180,E1 22119.22,E2 22119.22} C_VEL
LIN {X 0,Y 264.141,Z 1040.717,A -85,B 0,C 180,E1 22123.939,E2 22123.939} C_VEL
LIN {X 0,Y 266.568,Z 1030.995,A -85,B 0,C 180,E1 22130.223,E2 22130.223} C_VEL
LIN {X 0,Y 268.08,Z 1025.602,A -85,B 0,C 180,E1 22136.774,E2 22136.774} C_VEL
LIN {X 0,Y 268.671,Z 1024.818,A -85,B 0,C 180,E1 22140,E2 22140} C_VEL
LIN {X 0,Y 268.491,Z 1027.197,A -85,B 0,C 180,E1 22144.838,E2 22144.838} C_VEL
LIN {X 0,Y 268.027,Z 1034.627,A -85,B 0,C 180,E1 22151.365,E2 22151.365} C_VEL
LIN {X 0,Y 266.855,Z 1040.712,A -85,B 0,C 180,E1 22154.612,E2 22154.612} C_VEL
LIN {X 0,Y 241.158,Z 1072.862,A -85,B 0,C 180,E1 22158.766,E2 22158.766} C_VEL
LIN {X 0,Y 214.257,Z 1100.838,A -85,B 0,C 180,E1 22164.667,E2 22164.667} C_VEL
LIN {X 0,Y 188.422,Z 1123.931,A -85,B 0,C 180,E1 22172.764,E2 22172.764} C_VEL
LIN {X 0,Y 164.697,Z 1143.233,A -85,B 0,C 180,E1 22184.759,E2 22184.759} C_VEL
LIN {X 0,Y 149.042,Z 1156.215,A -85,B 0,C 180,E1 22199.587,E2 22199.587} C_VEL
LIN {X 0,Y 143.397,Z 1162.04,A -85,B 0,C 180,E1 22211.598,E2 22211.598} C_VEL
LIN {X 0,Y 141.572,Z 1164.956,A -85,B 0,C 180,E1 22223.882,E2 22223.882} C_VEL
LIN {X 0,Y 141.893,Z 1165.342,A -85,B 0,C 180,E1 22230.001,E2 22230.001} C_VEL
LIN {X 0,Y 141.975,Z 1163.865,A -85,B 0,C 180,E1 22242.274,E2 22242.274} C_VEL
LIN {X 0,Y 147.16,Z 1157.896,A -85,B 0,C 180,E1 22257.481,E2 22257.481} C_VEL
LIN {X 0,Y 161.155,Z 1146.04,A -85,B 0,C 180,E1 22272.756,E2 22272.756} C_VEL
LIN {X 0,Y 181.541,Z 1129.703,A -85,B 0,C 180,E1 22284.42,E2 22284.42} C_VEL
LIN {X 0,Y 207.846,Z 1107.007,A -85,B 0,C 180,E1 22293.63,E2 22293.63} C_VEL
LIN {X 0,Y 236.065,Z 1078.865,A -85,B 0,C 180,E1 22300.208,E2 22300.208} C_VEL
LIN {X 0,Y 262.898,Z 1046.469,A -85,B 0,C 180,E1 22304.803,E2 22304.803} C_VEL
LIN {X 0,Y 266.971,Z 1040.807,A -85,B 0,C 180,E1 22305.389,E2 22305.389} C_VEL
LIN {X 0,Y 268.29,Z 1033.501,A -85,B 0,C 180,E1 22309.467,E2 22309.467} C_VEL
LIN {X 0,Y 268.74,Z 1026.179,A -85,B 0,C 180,E1 22316.781,E2 22316.781} C_VEL
LIN {X 0,Y 268.786,Z 1024.993,A -85,B 0,C 180,E1 22320,E2 22320} C_VEL
LIN {X 0,Y 267.757,Z 1026.805,A -85,B 0,C 180,E1 22324.834,E2 22324.834} C_VEL
LIN {X 0,Y 266.065,Z 1033.398,A -85,B 0,C 180,E1 22331.449,E2 22331.449} C_VEL
LIN {X 0,Y 263.938,Z 1041.378,A -85,B 0,C 180,E1 22336.135,E2 22336.135} C_VEL
LIN {X 0,Y 237.826,Z 1072.52,A -85,B 0,C 180,E1 22340.755,E2 22340.755} C_VEL
LIN {X 0,Y 209.584,Z 1100.139,A -85,B 0,C 180,E1 22347.463,E2 22347.463} C_VEL
LIN {X 0,Y 183.312,Z 1121.95,A -85,B 0,C 180,E1 22356.618,E2 22356.618} C_VEL
LIN {X 0,Y 161.395,Z 1138.392,A -85,B 0,C 180,E1 22369.118,E2 22369.118} C_VEL
LIN {X 0,Y 148.563,Z 1148.066,A -85,B 0,C 180,E1 22382.8,E2 22382.8} C_VEL
LIN {X 0,Y 146.307,Z 1149.951,A -85,B 0,C 180,E1 22386.765,E2 22386.765} C_VEL
LIN {X 0,Y 141.647,Z 1151.989,A -85,B 0,C 180,E1 22391.57,E2 22391.57} C_VEL
LIN {X 0,Y 134.37,Z 1154.063,A -85,B 0,C 180,E1 22399.186,E2 22399.186} C_VEL
LIN {X 0,Y 134.15,Z 1154.198,A -85,B 0,C 180,E1 22400.118,E2 22400.118} C_VEL
LIN {X 0,Y 134.104,Z 1154.992,A -85,B 0,C 180,E1 22409.999,E2 22409.999} C_VEL
LIN {X 0,Y 134.742,Z 1153.717,A -85,B 0,C 180,E1 22422.943,E2 22422.943} C_VEL
LIN {X 0,Y 141.437,Z 1148.299,A -85,B 0,C 180,E1 22438.692,E2 22438.692} C_VEL
LIN {X 0,Y 155.428,Z 1138.575,A -85,B 0,C 180,E1 22452.813,E2 22452.813} C_VEL
LIN {X 0,Y 178.688,Z 1122.089,A -85,B 0,C 180,E1 22465.424,E2 22465.424} C_VEL
LIN {X 0,Y 206.637,Z 1099.701,A -85,B 0,C 180,E1 22474.649,E2 22474.649} C_VEL
LIN {X 0,Y 234.619,Z 1073.115,A -85,B 0,C 180,E1 22480.93,E2 22480.93} C_VEL
LIN {X 0,Y 259.207,Z 1044.508,A -85,B 0,C 180,E1 22485.259,E2 22485.259} C_VEL
LIN {X 0,Y 261.661,Z 1036.203,A -85,B 0,C 180,E1 22491.197,E2 22491.197} C_VEL
LIN {X 0,Y 263.264,Z 1031.976,A -85,B 0,C 180,E1 22496.714,E2 22496.714} C_VEL
LIN {X 0,Y 263.923,Z 1031.16,A -85,B 0,C 180,E1 22500,E2 22500} C_VEL
LIN {X 0,Y 263.629,Z 1033.623,A -85,B 0,C 180,E1 22504.926,E2 22504.926} C_VEL
LIN {X 0,Y 262.885,Z 1039.962,A -85,B 0,C 180,E1 22510.753,E2 22510.753} C_VEL
LIN {X 0,Y 261.995,Z 1044.434,A -85,B 0,C 180,E1 22513.32,E2 22513.32} C_VEL
LIN {X 0,Y 233.764,Z 1077.961,A -85,B 0,C 180,E1 22517.796,E2 22517.796} C_VEL
LIN {X 0,Y 203.906,Z 1106.936,A -85,B 0,C 180,E1 22524.395,E2 22524.395} C_VEL
LIN {X 0,Y 176.488,Z 1129.668,A -85,B 0,C 180,E1 22533.609,E2 22533.609} C_VEL
LIN {X 0,Y 153.382,Z 1147.052,A -85,B 0,C 180,E1 22546.475,E2 22546.475} C_VEL
LIN {X 0,Y 139.807,Z 1157.701,A -85,B 0,C 180,E1 22561.244,E2 22561.244} C_VEL
LIN {X 0,Y 134.174,Z 1163.553,A -85,B 0,C 180,E1 22577.002,E2 22577.002} C_VEL
LIN {X 0,Y 133.98,Z 1165.045,A -85,B 0,C 180,E1 22590.001,E2 22590.001} C_VEL
LIN {X 0,Y 134.157,Z 1163.565,A -85,B 0,C 180,E1 22603.001,E2 22603.001} C_VEL
LIN {X 0,Y 139.811,Z 1157.728,A -85,B 0,C 180,E1 22618.762,E2 22618.762} C_VEL
LIN {X 0,Y 155.208,Z 1145.732,A -85,B 0,C 180,E1 22634.821,E2 22634.821} C_VEL
LIN {X 0,Y 177.625,Z 1128.786,A -85,B 0,C 180,E1 22646.902,E2 22646.902} C_VEL
LIN {X 0,Y 205.662,Z 1105.461,A -85,B 0,C 180,E1 22656.055,E2 22656.055} C_VEL
LIN {X 0,Y 233.819,Z 1078.137,A -85,B 0,C 180,E1 22662.164,E2 22662.164} C_VEL
LIN {X 0,Y 260.886,Z 1046.173,A -85,B 0,C 180,E1 22666.522,E2 22666.522} C_VEL
LIN {X 0,Y 262.04,Z 1044.618,A -85,B 0,C 180,E1 22666.683,E2 22666.683} C_VEL
LIN {X 0,Y 263.166,Z 1038.888,A -85,B 0,C 180,E1 22670.095,E2 22670.095} C_VEL
LIN {X 0,Y 263.935,Z 1032.583,A -85,B 0,C 180,E1 22676.722,E2 22676.722} C_VEL
LIN {X 0,Y 264.044,Z 1031.326,A -85,B 0,C 180,E1 22680,E2 22680} C_VEL
LIN {X 0,Y 262.832,Z 1033.196,A -85,B 0,C 180,E1 22684.94,E2 22684.94} C_VEL
LIN {X 0,Y 261.091,Z 1038.71,A -85,B 0,C 180,E1 22690.72,E2 22690.72} C_VEL
LIN {X 0,Y 259.414,Z 1044.46,A -85,B 0,C 180,E1 22694.607,E2 22694.607} C_VEL
LIN {X 0,Y 232.687,Z 1075.228,A -85,B 0,C 180,E1 22699.36,E2 22699.36} C_VEL
LIN {X 0,Y 205.115,Z 1101.138,A -85,B 0,C 180,E1 22705.68,E2 22705.68} C_VEL
LIN {X 0,Y 178.545,Z 1122.256,A -85,B 0,C 180,E1 22714.507,E2 22714.507} C_VEL
LIN {X 0,Y 155.338,Z 1138.696,A -85,B 0,C 180,E1 22727.155,E2 22727.155} C_VEL
LIN {X 0,Y 139.538,Z 1149.85,A -85,B 0,C 180,E1 22744.368,E2 22744.368} C_VEL
LIN {X 0,Y 134.15,Z 1154.198,A -85,B 0,C 180,E1 22760.118,E2 22760.118} C_VEL
LIN {X 0,Y 131.204,Z 1154.933,A -85,B 0,C 180,E1 22765.649,E2 22765.649} C_VEL
LIN {X 0,Y 125.952,Z 1155.048,A -85,B 0,C 180,E1 22775.329,E2 22775.329} C_VEL
LIN {X 0,Y 129.315,Z 1152.226,A -85,B 0,C 180,E1 22791.014,E2 22791.014} C_VEL
LIN {X 0,Y 142.547,Z 1143.367,A -85,B 0,C 180,E1 22809.431,E2 22809.431} C_VEL
LIN {X 0,Y 164.546,Z 1129.049,A -85,B 0,C 180,E1 22823.518,E2 22823.518} C_VEL
LIN {X 0,Y 192.31,Z 1108.902,A -85,B 0,C 180,E1 22833.771,E2 22833.771} C_VEL
LIN {X 0,Y 223.247,Z 1082.151,A -85,B 0,C 180,E1 22841.139,E2 22841.139} C_VEL
LIN {X 0,Y 251.589,Z 1052.008,A -85,B 0,C 180,E1 22845.976,E2 22845.976} C_VEL
LIN {X 0,Y 254.346,Z 1048.279,A -85,B 0,C 180,E1 22846.71,E2 22846.71} C_VEL
LIN {X 0,Y 257.009,Z 1040.895,A -85,B 0,C 180,E1 22852.764,E2 22852.764} C_VEL
LIN {X 0,Y 258.173,Z 1038.181,A -85,B 0,C 180,E1 22856.65,E2 22856.65} C_VEL
LIN {X 0,Y 258.937,Z 1037.287,A -85,B 0,C 180,E1 22860,E2 22860} C_VEL
LIN {X 0,Y 258.513,Z 1039.872,A -85,B 0,C 180,E1 22865.025,E2 22865.025} C_VEL
LIN {X 0,Y 257.397,Z 1046.919,A -85,B 0,C 180,E1 22871.229,E2 22871.229} C_VEL
LIN {X 0,Y 256.359,Z 1049.047,A -85,B 0,C 180,E1 22872.089,E2 22872.089} C_VEL
LIN {X 0,Y 229.761,Z 1079.327,A -85,B 0,C 180,E1 22876.152,E2 22876.152} C_VEL
LIN {X 0,Y 199.463,Z 1107.591,A -85,B 0,C 180,E1 22882.547,E2 22882.547} C_VEL
LIN {X 0,Y 171.912,Z 1129.46,A -85,B 0,C 180,E1 22891.369,E2 22891.369} C_VEL
LIN {X 0,Y 147.526,Z 1146.742,A -85,B 0,C 180,E1 22904.274,E2 22904.274} C_VEL
LIN {X 0,Y 132.557,Z 1157.505,A -85,B 0,C 180,E1 22919.767,E2 22919.767} C_VEL
LIN {X 0,Y 126.364,Z 1163.252,A -85,B 0,C 180,E1 22936.183,E2 22936.183} C_VEL
LIN {X 0,Y 126.062,Z 1164.748,A -85,B 0,C 180,E1 22950.001,E2 22950.001} C_VEL
LIN {X 0,Y 126.346,Z 1163.264,A -85,B 0,C 180,E1 22963.821,E2 22963.821} C_VEL
LIN {X 0,Y 132.562,Z 1157.535,A -85,B 0,C 180,E1 22980.236,E2 22980.236} C_VEL
LIN {X 0,Y 147.538,Z 1146.8,A -85,B 0,C 180,E1 22995.723,E2 22995.723} C_VEL
LIN {X 0,Y 173.218,Z 1128.493,A -85,B 0,C 180,E1 23009.191,E2 23009.191} C_VEL
LIN {X 0,Y 202.866,Z 1104.795,A -85,B 0,C 180,E1 23018.282,E2 23018.282} C_VEL
LIN {X 0,Y 231.438,Z 1077.832,A -85,B 0,C 180,E1 23024.098,E2 23024.098} C_VEL
LIN {X 0,Y 257.307,Z 1047.911,A -85,B 0,C 180,E1 23028.193,E2 23028.193} C_VEL
LIN {X 0,Y 258.353,Z 1041.565,A -85,B 0,C 180,E1 23033.291,E2 23033.291} C_VEL
LIN {X 0,Y 258.84,Z 1038.797,A -85,B 0,C 180,E1 23036.658,E2 23036.658} C_VEL
LIN {X 0,Y 259.036,Z 1037.464,A -85,B 0,C 180,E1 23040,E2 23040} C_VEL
LIN {X 0,Y 257.629,Z 1039.629,A -85,B 0,C 180,E1 23045.285,E2 23045.285} C_VEL
LIN {X 0,Y 255.6,Z 1045.18,A -85,B 0,C 180,E1 23050.953,E2 23050.953} C_VEL
LIN {X 0,Y 254.432,Z 1048.5,A -85,B 0,C 180,E1 23053.286,E2 23053.286} C_VEL
LIN {X 0,Y 228.075,Z 1077.541,A -85,B 0,C 180,E1 23057.836,E2 23057.836} C_VEL
LIN {X 0,Y 200.243,Z 1102.615,A -85,B 0,C 180,E1 23063.973,E2 23063.973} C_VEL
LIN {X 0,Y 171.534,Z 1124.272,A -85,B 0,C 180,E1 23073.307,E2 23073.307} C_VEL
LIN {X 0,Y 147.599,Z 1140.158,A -85,B 0,C 180,E1 23086.361,E2 23086.361} C_VEL
LIN {X 0,Y 132.324,Z 1150.152,A -85,B 0,C 180,E1 23102.86,E2 23102.86} C_VEL
LIN {X 0,Y 126.254,Z 1154.555,A -85,B 0,C 180,E1 23119.924,E2 23119.924} C_VEL
LIN {X 0,Y 126.193,Z 1155.288,A -85,B 0,C 180,E1 23129.999,E2 23129.999} C_VEL
LIN {X 0,Y 125.952,Z 1155.048,A -85,B 0,C 180,E1 23135.329,E2 23135.329} C_VEL
LIN {X 0,Y 124.003,Z 1154.56,A -85,B 0,C 180,E1 23141.266,E2 23141.266} C_VEL
LIN {X 0,Y 121.115,Z 1153.01,A -85,B 0,C 180,E1 23150.467,E2 23150.467} C_VEL
LIN {X 0,Y 121.47,Z 1152.773,A -85,B 0,C 180,E1 23151.491,E2 23151.491} C_VEL
LIN {X 0,Y 133.064,Z 1145.539,A -85,B 0,C 180,E1 23168.629,E2 23168.629} C_VEL
LIN {X 0,Y 155.227,Z 1132.181,A -85,B 0,C 180,E1 23183.716,E2 23183.716} C_VEL
LIN {X 0,Y 181.867,Z 1114.34,A -85,B 0,C 180,E1 23193.925,E2 23193.925} C_VEL
LIN {X 0,Y 210.155,Z 1091.993,A -85,B 0,C 180,E1 23201.062,E2 23201.062} C_VEL
LIN {X 0,Y 240.585,Z 1062.563,A -85,B 0,C 180,E1 23206.457,E2 23206.457} C_VEL
LIN {X 0,Y 249.069,Z 1053.123,A -85,B 0,C 180,E1 23207.671,E2 23207.671} C_VEL
LIN {X 0,Y 251.804,Z 1046.627,A -85,B 0,C 180,E1 23213.117,E2 23213.117} C_VEL
LIN {X 0,Y 253.013,Z 1044.342,A -85,B 0,C 180,E1 23216.581,E2 23216.581} C_VEL
LIN {X 0,Y 253.901,Z 1043.41,A -85,B 0,C 180,E1 23220,E2 23220} C_VEL
LIN {X 0,Y 253.316,Z 1046.063,A -85,B 0,C 180,E1 23225.128,E2 23225.128} C_VEL
LIN {X 0,Y 252.118,Z 1051.674,A -85,B 0,C 180,E1 23230.344,E2 23230.344} C_VEL
LIN {X 0,Y 248.959,Z 1055.837,A -85,B 0,C 180,E1 23231.038,E2 23231.038} C_VEL
LIN {X 0,Y 219.354,Z 1087.114,A -85,B 0,C 180,E1 23235.613,E2 23235.613} C_VEL
LIN {X 0,Y 187.885,Z 1114.206,A -85,B 0,C 180,E1 23242.538,E2 23242.538} C_VEL
LIN {X 0,Y 157.64,Z 1136.085,A -85,B 0,C 180,E1 23253.114,E2 23253.114} C_VEL
LIN {X 0,Y 134.441,Z 1151.247,A -85,B 0,C 180,E1 23267.666,E2 23267.666} C_VEL
LIN {X 0,Y 121.993,Z 1159.863,A -85,B 0,C 180,E1 23284.347,E2 23284.347} C_VEL
LIN {X 0,Y 117.834,Z 1164.059,A -85,B 0,C 180,E1 23302.643,E2 23302.643} C_VEL
LIN {X 0,Y 118.159,Z 1164.452,A -85,B 0,C 180,E1 23310.001,E2 23310.001} C_VEL
LIN {X 0,Y 118.564,Z 1162.964,A -85,B 0,C 180,E1 23324.748,E2 23324.748} C_VEL
LIN {X 0,Y 123.759,Z 1158.603,A -85,B 0,C 180,E1 23339.192,E2 23339.192} C_VEL
LIN {X 0,Y 141.911,Z 1146.492,A -85,B 0,C 180,E1 23358.104,E2 23358.104} C_VEL
LIN {X 0,Y 167.945,Z 1129.053,A -85,B 0,C 180,E1 23371.167,E2 23371.167} C_VEL
LIN {X 0,Y 199.048,Z 1105.287,A -85,B 0,C 180,E1 23380.258,E2 23380.258} C_VEL
LIN {X 0,Y 229.326,Z 1077.527,A -85,B 0,C 180,E1 23386.07,E2 23386.07} C_VEL
LIN {X 0,Y 251.185,Z 1053.323,A -85,B 0,C 180,E1 23389.268,E2 23389.268} C_VEL
LIN {X 0,Y 252.228,Z 1051.78,A -85,B 0,C 180,E1 23389.66,E2 23389.66} C_VEL
LIN {X 0,Y 253.702,Z 1044.976,A -85,B 0,C 180,E1 23396.59,E2 23396.59} C_VEL
LIN {X 0,Y 253.994,Z 1043.585,A -85,B 0,C 180,E1 23400,E2 23400} C_VEL
LIN {X 0,Y 252.357,Z 1045.773,A -85,B 0,C 180,E1 23405.396,E2 23405.396} C_VEL
LIN {X 0,Y 249.838,Z 1051.833,A -85,B 0,C 180,E1 23411.382,E2 23411.382} C_VEL
LIN {X 0,Y 248.973,Z 1053.425,A -85,B 0,C 180,E1 23412.224,E2 23412.224} C_VEL
LIN {X 0,Y 219.566,Z 1083.76,A -85,B 0,C 180,E1 23417.021,E2 23417.021} C_VEL
LIN {X 0,Y 189.092,Z 1109.145,A -85,B 0,C 180,E1 23423.859,E2 23423.859} C_VEL
LIN {X 0,Y 159.422,Z 1129.687,A -85,B 0,C 180,E1 23434.24,E2 23434.24} C_VEL
LIN {X 0,Y 136.294,Z 1143.772,A -85,B 0,C 180,E1 23448.37,E2 23448.37} C_VEL
LIN {X 0,Y 123.194,Z 1151.604,A -85,B 0,C 180,E1 23464.613,E2 23464.613} C_VEL
LIN {X 0,Y 118.198,Z 1155.291,A -85,B 0,C 180,E1 23482.664,E2 23482.664} C_VEL
LIN {X 0,Y 118.284,Z 1155.585,A -85,B 0,C 180,E1 23489.999,E2 23489.999} C_VEL
LIN {X 0,Y 119.243,Z 1154.316,A -85,B 0,C 180,E1 23504.66,E2 23504.66} C_VEL
LIN {X 0,Y 121.47,Z 1152.773,A -85,B 0,C 180,E1 23511.491,E2 23511.491} C_VEL
LIN {X 0,Y 122.048,Z 1151.304,A -85,B 0,C 180,E1 23517.616,E2 23517.616} C_VEL
LIN {X 0,Y 122.973,Z 1148.124,A -85,B 0,C 180,E1 23526.809,E2 23526.809} C_VEL
LIN {X 0,Y 123.7,Z 1147.634,A -85,B 0,C 180,E1 23527.75,E2 23527.75} C_VEL
LIN {X 0,Y 145.279,Z 1135.625,A -85,B 0,C 180,E1 23543.609,E2 23543.609} C_VEL
LIN {X 0,Y 176.072,Z 1116.347,A -85,B 0,C 180,E1 23555.584,E2 23555.584} C_VEL
LIN {X 0,Y 206.969,Z 1092.89,A -85,B 0,C 180,E1 23563.045,E2 23563.045} C_VEL
LIN {X 0,Y 238.24,Z 1063.512,A -85,B 0,C 180,E1 23568.254,E2 23568.254} C_VEL
LIN {X 0,Y 243.959,Z 1057.256,A -85,B 0,C 180,E1 23569.031,E2 23569.031} C_VEL
LIN {X 0,Y 246.303,Z 1052.772,A -85,B 0,C 180,E1 23572.982,E2 23572.982} C_VEL
LIN {X 0,Y 247.627,Z 1050.333,A -85,B 0,C 180,E1 23576.507,E2 23576.507} C_VEL
LIN {X 0,Y 248.603,Z 1049.311,A -85,B 0,C 180,E1 23580,E2 23580} C_VEL
LIN {X 0,Y 247.899,Z 1052.101,A -85,B 0,C 180,E1 23585.239,E2 23585.239} C_VEL
LIN {X 0,Y 246.574,Z 1056.651,A -85,B 0,C 180,E1 23589.312,E2 23589.312} C_VEL
LIN {X 0,Y 216.13,Z 1087.897,A -85,B 0,C 180,E1 23593.727,E2 23593.727} C_VEL
LIN {X 0,Y 183.324,Z 1115.029,A -85,B 0,C 180,E1 23600.558,E2 23600.558} C_VEL
LIN {X 0,Y 153.283,Z 1135.774,A -85,B 0,C 180,E1 23610.526,E2 23610.526} C_VEL
LIN {X 0,Y 128.477,Z 1150.937,A -85,B 0,C 180,E1 23625.193,E2 23625.193} C_VEL
LIN {X 0,Y 114.717,Z 1159.557,A -85,B 0,C 180,E1 23642.588,E2 23642.588} C_VEL
LIN {X 0,Y 109.926,Z 1163.76,A -85,B 0,C 180,E1 23662.111,E2 23662.111} C_VEL
LIN {X 0,Y 110.236,Z 1164.155,A -85,B 0,C 180,E1 23670.001,E2 23670.001} C_VEL
LIN {X 0,Y 110.805,Z 1162.662,A -85,B 0,C 180,E1 23685.806,E2 23685.806} C_VEL
LIN {X 0,Y 116.687,Z 1158.297,A -85,B 0,C 180,E1 23701.151,E2 23701.151} C_VEL
LIN {X 0,Y 136.537,Z 1146.184,A -85,B 0,C 180,E1 23720.683,E2 23720.683} C_VEL
LIN {X 0,Y 164.519,Z 1128.455,A -85,B 0,C 180,E1 23733.844,E2 23733.844} C_VEL
LIN {X 0,Y 196.483,Z 1104.927,A -85,B 0,C 180,E1 23742.532,E2 23742.532} C_VEL
LIN {X 0,Y 227.49,Z 1077.222,A -85,B 0,C 180,E1 23748.076,E2 23748.076} C_VEL
LIN {X 0,Y 246.566,Z 1056.859,A -85,B 0,C 180,E1 23750.704,E2 23750.704} C_VEL
LIN {X 0,Y 247.592,Z 1053.869,A -85,B 0,C 180,E1 23752.998,E2 23752.998} C_VEL
LIN {X 0,Y 248.324,Z 1050.958,A -85,B 0,C 180,E1 23756.516,E2 23756.516} C_VEL
LIN {X 0,Y 248.681,Z 1049.492,A -85,B 0,C 180,E1 23760,E2 23760} C_VEL
LIN {X 0,Y 247.031,Z 1051.638,A -85,B 0,C 180,E1 23765.257,E2 23765.257} C_VEL
LIN {X 0,Y 244.485,Z 1056.814,A -85,B 0,C 180,E1 23770.67,E2 23770.67} C_VEL
LIN {X 0,Y 214.837,Z 1086.211,A -85,B 0,C 180,E1 23775.409,E2 23775.409} C_VEL
LIN {X 0,Y 183.898,Z 1110.872,A -85,B 0,C 180,E1 23782.09,E2 23782.09} C_VEL
LIN {X 0,Y 155.402,Z 1129.754,A -85,B 0,C 180,E1 23791.575,E2 23791.575} C_VEL
LIN {X 0,Y 130.324,Z 1144.076,A -85,B 0,C 180,E1 23805.993,E2 23805.993} C_VEL
LIN {X 0,Y 115.978,Z 1151.905,A -85,B 0,C 180,E1 23822.909,E2 23822.909} C_VEL
LIN {X 0,Y 110.315,Z 1155.589,A -85,B 0,C 180,E1 23842.137,E2 23842.137} C_VEL
LIN {X 0,Y 110.372,Z 1155.882,A -85,B 0,C 180,E1 23849.999,E2 23849.999} C_VEL
LIN {X 0,Y 111.53,Z 1154.616,A -85,B 0,C 180,E1 23865.699,E2 23865.699} C_VEL
LIN {X 0,Y 120.694,Z 1149.212,A -85,B 0,C 180,E1 23884.237,E2 23884.237} C_VEL
LIN {X 0,Y 123.7,Z 1147.634,A -85,B 0,C 180,E1 23887.75,E2 23887.75} C_VEL
LIN {X 0,Y 127.662,Z 1144.059,A -85,B 0,C 180,E1 23895.377,E2 23895.377} C_VEL
LIN {X 0,Y 133.412,Z 1139.768,A -85,B 0,C 180,E1 23902.422,E2 23902.422} C_VEL
LIN {X 0,Y 162.261,Z 1123.396,A -85,B 0,C 180,E1 23914.936,E2 23914.936} C_VEL
LIN {X 0,Y 194.942,Z 1100.93,A -85,B 0,C 180,E1 23923.32,E2 23923.32} C_VEL
LIN {X 0,Y 227.256,Z 1073.229,A -85,B 0,C 180,E1 23928.858,E2 23928.858} C_VEL
LIN {X 0,Y 238.133,Z 1062.311,A -85,B 0,C 180,E1 23930.342,E2 23930.342} C_VEL
LIN {X 0,Y 239.545,Z 1060.622,A -85,B 0,C 180,E1 23930.843,E2 23930.843} C_VEL
LIN {X 0,Y 242.145,Z 1056.242,A -85,B 0,C 180,E1 23936.428,E2 23936.428} C_VEL
LIN {X 0,Y 243.283,Z 1055.182,A -85,B 0,C 180,E1 23940,E2 23940} C_VEL
LIN {X 0,Y 242.414,Z 1057.873,A -85,B 0,C 180,E1 23945.135,E2 23945.135} C_VEL
LIN {X 0,Y 241.703,Z 1060.166,A -85,B 0,C 180,E1 23947.623,E2 23947.623} C_VEL
LIN {X 0,Y 234.186,Z 1068.395,A -85,B 0,C 180,E1 23948.768,E2 23948.768} C_VEL
LIN {X 0,Y 201.888,Z 1098.238,A -85,B 0,C 180,E1 23953.669,E2 23953.669} C_VEL
LIN {X 0,Y 170.306,Z 1121.948,A -85,B 0,C 180,E1 23960.758,E2 23960.758} C_VEL
LIN {X 0,Y 138.709,Z 1141.657,A -85,B 0,C 180,E1 23972.495,E2 23972.495} C_VEL
LIN {X 0,Y 115.517,Z 1154.672,A -85,B 0,C 180,E1 23989.221,E2 23989.221} C_VEL
LIN {X 0,Y 105.722,Z 1160.518,A -85,B 0,C 180,E1 24004.647,E2 24004.647} C_VEL
LIN {X 0,Y 102.046,Z 1163.461,A -85,B 0,C 180,E1 24021.497,E2 24021.497} C_VEL
LIN {X 0,Y 102.321,Z 1163.858,A -85,B 0,C 180,E1 24030.001,E2 24030.001} C_VEL
LIN {X 0,Y 103.107,Z 1162.362,A -85,B 0,C 180,E1 24047.021,E2 24047.021} C_VEL
LIN {X 0,Y 113.081,Z 1156.015,A -85,B 0,C 180,E1 24067.936,E2 24067.936} C_VEL
LIN {X 0,Y 134.132,Z 1144.302,A -85,B 0,C 180,E1 24085.047,E2 24085.047} C_VEL
LIN {X 0,Y 163.588,Z 1126.443,A -85,B 0,C 180,E1 24097.288,E2 24097.288} C_VEL
LIN {X 0,Y 195.23,Z 1103.761,A -85,B 0,C 180,E1 24105.057,E2 24105.057} C_VEL
LIN {X 0,Y 227.593,Z 1075.232,A -85,B 0,C 180,E1 24110.354,E2 24110.354} C_VEL
LIN {X 0,Y 241.869,Z 1060.214,A -85,B 0,C 180,E1 24112.382,E2 24112.382} C_VEL
LIN {X 0,Y 242.859,Z 1056.893,A -85,B 0,C 180,E1 24116.437,E2 24116.437} C_VEL
LIN {X 0,Y 243.349,Z 1055.359,A -85,B 0,C 180,E1 24120,E2 24120} C_VEL
LIN {X 0,Y 241.413,Z 1057.56,A -85,B 0,C 180,E1 24125.378,E2 24125.378} C_VEL
LIN {X 0,Y 239.644,Z 1060.756,A -85,B 0,C 180,E1 24129.081,E2 24129.081} C_VEL
LIN {X 0,Y 231.605,Z 1069.116,A -85,B 0,C 180,E1 24130.446,E2 24130.446} C_VEL
LIN {X 0,Y 201.333,Z 1096.025,A -85,B 0,C 180,E1 24135.333,E2 24135.333} C_VEL
LIN {X 0,Y 171.267,Z 1117.778,A -85,B 0,C 180,E1 24142.309,E2 24142.309} C_VEL
LIN {X 0,Y 140.485,Z 1136.046,A -85,B 0,C 180,E1 24153.646,E2 24153.646} C_VEL
LIN {X 0,Y 117.22,Z 1148.084,A -85,B 0,C 180,E1 24169.933,E2 24169.933} C_VEL
LIN {X 0,Y 106.854,Z 1153.338,A -85,B 0,C 180,E1 24184.933,E2 24184.933} C_VEL
LIN {X 0,Y 102.441,Z 1155.887,A -85,B 0,C 180,E1 24201.528,E2 24201.528} C_VEL
LIN {X 0,Y 102.479,Z 1156.178,A -85,B 0,C 180,E1 24209.999,E2 24209.999} C_VEL
LIN {X 0,Y 103.86,Z 1154.916,A -85,B 0,C 180,E1 24226.892,E2 24226.892} C_VEL
LIN {X 0,Y 113.487,Z 1149.817,A -85,B 0,C 180,E1 24245.799,E2 24245.799} C_VEL
LIN {X 0,Y 133.412,Z 1139.768,A -85,B 0,C 180,E1 24262.422,E2 24262.422} C_VEL
LIN {X 0,Y 140.696,Z 1134.868,A -85,B 0,C 180,E1 24268.779,E2 24268.779} C_VEL
LIN {X 0,Y 149.28,Z 1129.256,A -85,B 0,C 180,E1 24274.401,E2 24274.401} C_VEL
LIN {X 0,Y 182.604,Z 1108.509,A -85,B 0,C 180,E1 24283.583,E2 24283.583} C_VEL
LIN {X 0,Y 214.963,Z 1083.378,A -85,B 0,C 180,E1 24289.35,E2 24289.35} C_VEL
LIN {X 0,Y 234.415,Z 1065.124,A -85,B 0,C 180,E1 24292.139,E2 24292.139} C_VEL
LIN {X 0,Y 236.498,Z 1061.978,A -85,B 0,C 180,E1 24296.342,E2 24296.342} C_VEL
LIN {X 0,Y 237.712,Z 1060.83,A -85,B 0,C 180,E1 24300,E2 24300} C_VEL
LIN {X 0,Y 236.464,Z 1064.322,A -85,B 0,C 180,E1 24305.961,E2 24305.961} C_VEL
LIN {X 0,Y 233.469,Z 1067.708,A -85,B 0,C 180,E1 24306.743,E2 24306.743} C_VEL
LIN {X 0,Y 201.735,Z 1096.659,A -85,B 0,C 180,E1 24311.122,E2 24311.122} C_VEL
LIN {X 0,Y 167.569,Z 1121.638,A -85,B 0,C 180,E1 24318.128,E2 24318.128} C_VEL
LIN {X 0,Y 134.743,Z 1141.186,A -85,B 0,C 180,E1 24329.366,E2 24329.366} C_VEL
LIN {X 0,Y 109.416,Z 1154.362,A -85,B 0,C 180,E1 24346.404,E2 24346.404} C_VEL
LIN {X 0,Y 98.445,Z 1160.213,A -85,B 0,C 180,E1 24362.623,E2 24362.623} C_VEL
LIN {X 0,Y 94.153,Z 1163.162,A -85,B 0,C 180,E1 24380.778,E2 24380.778} C_VEL
LIN {X 0,Y 94.393,Z 1163.561,A -85,B 0,C 180,E1 24390.001,E2 24390.001} C_VEL
LIN {X 0,Y 95.437,Z 1162.06,A -85,B 0,C 180,E1 24408.436,E2 24408.436} C_VEL
LIN {X 0,Y 106.956,Z 1155.594,A -85,B 0,C 180,E1 24430.91,E2 24430.91} C_VEL
LIN {X 0,Y 129.568,Z 1143.993,A -85,B 0,C 180,E1 24448.048,E2 24448.048} C_VEL
LIN {X 0,Y 160.58,Z 1126.135,A -85,B 0,C 180,E1 24460.007,E2 24460.007} C_VEL
LIN {X 0,Y 193.269,Z 1103.454,A -85,B 0,C 180,E1 24467.419,E2 24467.419} C_VEL
LIN {X 0,Y 226.379,Z 1074.912,A -85,B 0,C 180,E1 24472.402,E2 24472.402} C_VEL
LIN {X 0,Y 235.118,Z 1066.247,A -85,B 0,C 180,E1 24473.46,E2 24473.46} C_VEL
LIN {X 0,Y 236.546,Z 1064.471,A -85,B 0,C 180,E1 24474.027,E2 24474.027} C_VEL
LIN {X 0,Y 237.768,Z 1061.016,A -85,B 0,C 180,E1 24480,E2 24480} C_VEL
LIN {X 0,Y 235.684,Z 1063.393,A -85,B 0,C 180,E1 24485.511,E2 24485.511} C_VEL
LIN {X 0,Y 234.554,Z 1065.239,A -85,B 0,C 180,E1 24487.857,E2 24487.857} C_VEL
LIN {X 0,Y 202.866,Z 1093.645,A -85,B 0,C 180,E1 24492.497,E2 24492.497} C_VEL
LIN {X 0,Y 168.342,Z 1118.082,A -85,B 0,C 180,E1 24499.742,E2 24499.742} C_VEL
LIN {X 0,Y 136.123,Z 1136.351,A -85,B 0,C 180,E1 24510.779,E2 24510.779} C_VEL
LIN {X 0,Y 111.119,Z 1148.388,A -85,B 0,C 180,E1 24527.233,E2 24527.233} C_VEL
LIN {X 0,Y 97.096,Z 1154.733,A -85,B 0,C 180,E1 24548.818,E2 24548.818} C_VEL
LIN {X 0,Y 94.562,Z 1156.475,A -85,B 0,C 180,E1 24569.999,E2 24569.999} C_VEL
LIN {X 0,Y 97.117,Z 1154.69,A -85,B 0,C 180,E1 24591.215,E2 24591.215} C_VEL
LIN {X 0,Y 111.151,Z 1148.315,A -85,B 0,C 180,E1 24612.75,E2 24612.75} C_VEL
LIN {X 0,Y 136.229,Z 1136.239,A -85,B 0,C 180,E1 24629.144,E2 24629.144} C_VEL
LIN {X 0,Y 149.28,Z 1129.256,A -85,B 0,C 180,E1 24634.401,E2 24634.401} C_VEL
LIN {X 0,Y 158.958,Z 1123.006,A -85,B 0,C 180,E1 24639.315,E2 24639.315} C_VEL
LIN {X 0,Y 169.211,Z 1116.115,A -85,B 0,C 180,E1 24643.678,E2 24643.678} C_VEL
LIN {X 0,Y 203.06,Z 1092.335,A -85,B 0,C 180,E1 24649.948,E2 24649.948} C_VEL
LIN {X 0,Y 227.902,Z 1070.759,A -85,B 0,C 180,E1 24653.311,E2 24653.311} C_VEL
LIN {X 0,Y 229.783,Z 1068.727,A -85,B 0,C 180,E1 24654.524,E2 24654.524} C_VEL
LIN {X 0,Y 232.085,Z 1066.455,A -85,B 0,C 180,E1 24660,E2 24660} C_VEL
LIN {X 0,Y 231.021,Z 1068.95,A -85,B 0,C 180,E1 24664.859,E2 24664.859} C_VEL
LIN {X 0,Y 198.65,Z 1097.617,A -85,B 0,C 180,E1 24669.063,E2 24669.063} C_VEL
LIN {X 0,Y 165.827,Z 1120.933,A -85,B 0,C 180,E1 24675.264,E2 24675.264} C_VEL
LIN {X 0,Y 131.104,Z 1140.767,A -85,B 0,C 180,E1 24686.113,E2 24686.113} C_VEL
LIN {X 0,Y 103.599,Z 1154.052,A -85,B 0,C 180,E1 24703.258,E2 24703.258} C_VEL
LIN {X 0,Y 91.291,Z 1159.907,A -85,B 0,C 180,E1 24720.273,E2 24720.273} C_VEL
LIN {X 0,Y 86.286,Z 1162.862,A -85,B 0,C 180,E1 24739.929,E2 24739.929} C_VEL
LIN {X 0,Y 86.462,Z 1163.263,A -85,B 0,C 180,E1 24750.001,E2 24750.001} C_VEL
LIN {X 0,Y 87.822,Z 1161.758,A -85,B 0,C 180,E1 24770.101,E2 24770.101} C_VEL
LIN {X 0,Y 99.876,Z 1155.751,A -85,B 0,C 180,E1 24792.837,E2 24792.837} C_VEL
LIN {X 0,Y 125.189,Z 1143.778,A -85,B 0,C 180,E1 24811.174,E2 24811.174} C_VEL
LIN {X 0,Y 157.965,Z 1125.829,A -85,B 0,C 180,E1 24822.804,E2 24822.804} C_VEL
LIN {X 0,Y 191.634,Z 1103.145,A -85,B 0,C 180,E1 24829.839,E2 24829.839} C_VEL
LIN {X 0,Y 224.789,Z 1075.25,A -85,B 0,C 180,E1 24834.38,E2 24834.38} C_VEL
LIN {X 0,Y 230.57,Z 1069.621,A -85,B 0,C 180,E1 24835.037,E2 24835.037} C_VEL
LIN {X 0,Y 231.419,Z 1068.31,A -85,B 0,C 180,E1 24836.261,E2 24836.261} C_VEL
LIN {X 0,Y 232.122,Z 1066.643,A -85,B 0,C 180,E1 24840,E2 24840} C_VEL
LIN {X 0,Y 229.514,Z 1069.343,A -85,B 0,C 180,E1 24846.053,E2 24846.053} C_VEL
LIN {X 0,Y 226.32,Z 1072.498,A -85,B 0,C 180,E1 24846.817,E2 24846.817} C_VEL
LIN {X 0,Y 193.401,Z 1099.821,A -85,B 0,C 180,E1 24851.483,E2 24851.483} C_VEL
LIN {X 0,Y 159.311,Z 1122.182,A -85,B 0,C 180,E1 24858.698,E2 24858.698} C_VEL
LIN {X 0,Y 129.35,Z 1137.946,A -85,B 0,C 180,E1 24868.958,E2 24868.958} C_VEL
LIN {X 0,Y 105.296,Z 1148.692,A -85,B 0,C 180,E1 24884.228,E2 24884.228} C_VEL
LIN {X 0,Y 92.519,Z 1153.941,A -85,B 0,C 180,E1 24900.704,E2 24900.704} C_VEL
LIN {X 0,Y 86.736,Z 1156.484,A -85,B 0,C 180,E1 24919.98,E2 24919.98} C_VEL
LIN {X 0,Y 86.645,Z 1156.771,A -85,B 0,C 180,E1 24929.999,E2 24929.999} C_VEL
LIN {X 0,Y 88.681,Z 1155.516,A -85,B 0,C 180,E1 24949.895,E2 24949.895} C_VEL
LIN {X 0,Y 101.466,Z 1150.138,A -85,B 0,C 180,E1 24971.964,E2 24971.964} C_VEL
LIN {X 0,Y 126.706,Z 1139.128,A -85,B 0,C 180,E1 24989.704,E2 24989.704} C_VEL
LIN {X 0,Y 156.682,Z 1123.639,A -85,B 0,C 180,E1 25000.525,E2 25000.525} C_VEL
LIN {X 0,Y 169.211,Z 1116.115,A -85,B 0,C 180,E1 25003.678,E2 25003.678} C_VEL
LIN {X 0,Y 180.075,Z 1108.6,A -85,B 0,C 180,E1 25007.499,E2 25007.499} C_VEL
LIN {X 0,Y 191.411,Z 1100.357,A -85,B 0,C 180,E1 25010.731,E2 25010.731} C_VEL
LIN {X 0,Y 222.75,Z 1075.164,A -85,B 0,C 180,E1 25014.845,E2 25014.845} C_VEL
LIN {X 0,Y 224.707,Z 1073.184,A -85,B 0,C 180,E1 25016.15,E2 25016.15} C_VEL
LIN {X 0,Y 226.243,Z 1071.864,A -85,B 0,C 180,E1 25020,E2 25020} C_VEL
LIN {X 0,Y 225.638,Z 1073.116,A -85,B 0,C 180,E1 25022.875,E2 25022.875} C_VEL
LIN {X 0,Y 222.723,Z 1076.081,A -85,B 0,C 180,E1 25023.658,E2 25023.658} C_VEL
LIN {X 0,Y 186.809,Z 1105.318,A -85,B 0,C 180,E1 25028.3,E2 25028.3} C_VEL
LIN {X 0,Y 152.385,Z 1127.408,A -85,B 0,C 180,E1 25035.094,E2 25035.094} C_VEL
LIN {X 0,Y 118.355,Z 1144.875,A -85,B 0,C 180,E1 25046.813,E2 25046.813} C_VEL
LIN {X 0,Y 90.27,Z 1157.037,A -85,B 0,C 180,E1 25068.037,E2 25068.037} C_VEL
LIN {X 0,Y 79.324,Z 1161.873,A -85,B 0,C 180,E1 25092.017,E2 25092.017} C_VEL
LIN {X 0,Y 78.529,Z 1162.966,A -85,B 0,C 180,E1 25110.001,E2 25110.001} C_VEL
LIN {X 0,Y 80.298,Z 1161.456,A -85,B 0,C 180,E1 25132.078,E2 25132.078} C_VEL
LIN {X 0,Y 94.005,Z 1155.443,A -85,B 0,C 180,E1 25156.251,E2 25156.251} C_VEL
LIN {X 0,Y 121.405,Z 1143.468,A -85,B 0,C 180,E1 25174.608,E2 25174.608} C_VEL
LIN {X 0,Y 152.386,Z 1127.509,A -85,B 0,C 180,E1 25184.909,E2 25184.909} C_VEL
LIN {X 0,Y 188.572,Z 1104.183,A -85,B 0,C 180,E1 25192.011,E2 25192.011} C_VEL
LIN {X 0,Y 222.979,Z 1076.061,A -85,B 0,C 180,E1 25196.334,E2 25196.334} C_VEL
LIN {X 0,Y 225.625,Z 1073.47,A -85,B 0,C 180,E1 25196.751,E2 25196.751} C_VEL
LIN {X 0,Y 226.278,Z 1072.054,A -85,B 0,C 180,E1 25200,E2 25200} C_VEL
LIN {X 0,Y 224.364,Z 1073.82,A -85,B 0,C 180,E1 25204.557,E2 25204.557} C_VEL
LIN {X 0,Y 222.202,Z 1075.852,A -85,B 0,C 180,E1 25205.145,E2 25205.145} C_VEL
LIN {X 0,Y 188.364,Z 1102.743,A -85,B 0,C 180,E1 25209.681,E2 25209.681} C_VEL
LIN {X 0,Y 153.033,Z 1124.696,A -85,B 0,C 180,E1 25216.825,E2 25216.825} C_VEL
LIN {X 0,Y 119.89,Z 1140.833,A -85,B 0,C 180,E1 25228.227,E2 25228.227} C_VEL
LIN {X 0,Y 91.825,Z 1151.969,A -85,B 0,C 180,E1 25248.901,E2 25248.901} C_VEL
LIN {X 0,Y 81.118,Z 1155.87,A -85,B 0,C 180,E1 25268.448,E2 25268.448} C_VEL
LIN {X 0,Y 78.725,Z 1157.068,A -85,B 0,C 180,E1 25289.999,E2 25289.999} C_VEL
LIN {X 0,Y 81.219,Z 1155.816,A -85,B 0,C 180,E1 25311.813,E2 25311.813} C_VEL
LIN {X 0,Y 95.597,Z 1150.443,A -85,B 0,C 180,E1 25335.212,E2 25335.212} C_VEL
LIN {X 0,Y 122.694,Z 1139.481,A -85,B 0,C 180,E1 25352.945,E2 25352.945} C_VEL
LIN {X 0,Y 155.123,Z 1123.387,A -85,B 0,C 180,E1 25363.624,E2 25363.624} C_VEL
LIN {X 0,Y 190.359,Z 1101.132,A -85,B 0,C 180,E1 25370.57,E2 25370.57} C_VEL
LIN {X 0,Y 191.411,Z 1100.357,A -85,B 0,C 180,E1 25370.731,E2 25370.731} C_VEL
LIN {X 0,Y 202.931,Z 1091.515,A -85,B 0,C 180,E1 25373.603,E2 25373.603} C_VEL
LIN {X 0,Y 212.905,Z 1083.385,A -85,B 0,C 180,E1 25375.915,E2 25375.915} C_VEL
LIN {X 0,Y 214.483,Z 1082.025,A -85,B 0,C 180,E1 25376.107,E2 25376.107} C_VEL
LIN {X 0,Y 219.026,Z 1078.137,A -85,B 0,C 180,E1 25377.039,E2 25377.039} C_VEL
LIN {X 0,Y 220.319,Z 1077.225,A -85,B 0,C 180,E1 25380,E2 25380} C_VEL
LIN {X 0,Y 219.937,Z 1077.855,A -85,B 0,C 180,E1 25381.607,E2 25381.607} C_VEL
LIN {X 0,Y 185.628,Z 1105.124,A -85,B 0,C 180,E1 25385.812,E2 25385.812} C_VEL
LIN {X 0,Y 150.285,Z 1127.189,A -85,B 0,C 180,E1 25392.09,E2 25392.09} C_VEL
LIN {X 0,Y 114.423,Z 1144.762,A -85,B 0,C 180,E1 25403.306,E2 25403.306} C_VEL
LIN {X 0,Y 84.361,Z 1156.73,A -85,B 0,C 180,E1 25424.317,E2 25424.317} C_VEL
LIN {X 0,Y 72.921,Z 1161.138,A -85,B 0,C 180,E1 25445.553,E2 25445.553} C_VEL
LIN {X 0,Y 70.622,Z 1162.669,A -85,B 0,C 180,E1 25470.001,E2 25470.001} C_VEL
LIN {X 0,Y 72.871,Z 1161.153,A -85,B 0,C 180,E1 25494.468,E2 25494.468} C_VEL
LIN {X 0,Y 88.528,Z 1155.136,A -85,B 0,C 180,E1 25520.091,E2 25520.091} C_VEL
LIN {X 0,Y 117.869,Z 1143.258,A -85,B 0,C 180,E1 25538.154,E2 25538.154} C_VEL
LIN {X 0,Y 150.261,Z 1127.307,A -85,B 0,C 180,E1 25547.904,E2 25547.904} C_VEL
LIN {X 0,Y 187.336,Z 1104.071,A -85,B 0,C 180,E1 25554.479,E2 25554.479} C_VEL
LIN {X 0,Y 219.962,Z 1078.039,A -85,B 0,C 180,E1 25558.36,E2 25558.36} C_VEL
LIN {X 0,Y 220.338,Z 1077.411,A -85,B 0,C 180,E1 25560,E2 25560} C_VEL
LIN {X 0,Y 219.078,Z 1078.301,A -85,B 0,C 180,E1 25562.835,E2 25562.835} C_VEL
LIN {X 0,Y 214.964,Z 1081.822,A -85,B 0,C 180,E1 25563.768,E2 25563.768} C_VEL
LIN {X 0,Y 181.028,Z 1107.085,A -85,B 0,C 180,E1 25568.155,E2 25568.155} C_VEL
LIN {X 0,Y 148.019,Z 1126.434,A -85,B 0,C 180,E1 25574.529,E2 25574.529} C_VEL
LIN {X 0,Y 113.317,Z 1142.295,A -85,B 0,C 180,E1 25585.987,E2 25585.987} C_VEL
LIN {X 0,Y 85.876,Z 1152.273,A -85,B 0,C 180,E1 25605.34,E2 25605.34} C_VEL
LIN {X 0,Y 73.816,Z 1156.144,A -85,B 0,C 180,E1 25625.866,E2 25625.866} C_VEL
LIN {X 0,Y 70.821,Z 1157.365,A -85,B 0,C 180,E1 25649.999,E2 25649.999} C_VEL
LIN {X 0,Y 73.838,Z 1156.117,A -85,B 0,C 180,E1 25674.124,E2 25674.124} C_VEL
LIN {X 0,Y 90.642,Z 1150.556,A -85,B 0,C 180,E1 25699.398,E2 25699.398} C_VEL
LIN {X 0,Y 116.328,Z 1141.032,A -85,B 0,C 180,E1 25715.235,E2 25715.235} C_VEL
LIN {X 0,Y 151.729,Z 1124.421,A -85,B 0,C 180,E1 25726.256,E2 25726.256} C_VEL
LIN {X 0,Y 188.877,Z 1101.672,A -85,B 0,C 180,E1 25732.943,E2 25732.943} C_VEL
LIN {X 0,Y 214.483,Z 1082.025,A -85,B 0,C 180,E1 25736.107,E2 25736.107} C_VEL
LIN {X 0,Y 214.927,Z 1081.633,A -85,B 0,C 180,E1 25737.053,E2 25737.053} C_VEL
LIN {X 0,Y 210.481,Z 1085.422,A -85,B 0,C 180,E1 25738.981,E2 25738.981} C_VEL
LIN {X 0,Y 196.348,Z 1096.637,A -85,B 0,C 180,E1 25741.886,E2 25741.886} C_VEL
LIN {X 0,Y 194.089,Z 1098.27,A -85,B 0,C 180,E1 25742.173,E2 25742.173} C_VEL
LIN {X 0,Y 159.613,Z 1120.813,A -85,B 0,C 180,E1 25746.935,E2 25746.935} C_VEL
LIN {X 0,Y 121.566,Z 1140.118,A -85,B 0,C 180,E1 25755.845,E2 25755.845} C_VEL
LIN {X 0,Y 88.516,Z 1153.124,A -85,B 0,C 180,E1 25771.528,E2 25771.528} C_VEL
LIN {X 0,Y 71.106,Z 1158.989,A -85,B 0,C 180,E1 25790.458,E2 25790.458} C_VEL
LIN {X 0,Y 62.806,Z 1161.962,A -85,B 0,C 180,E1 25816.099,E2 25816.099} C_VEL
LIN {X 0,Y 62.681,Z 1162.371,A -85,B 0,C 180,E1 25830.001,E2 25830.001} C_VEL
LIN {X 0,Y 65.594,Z 1160.85,A -85,B 0,C 180,E1 25857.396,E2 25857.396} C_VEL
LIN {X 0,Y 83.49,Z 1154.828,A -85,B 0,C 180,E1 25884.425,E2 25884.425} C_VEL
LIN {X 0,Y 115.042,Z 1142.948,A -85,B 0,C 180,E1 25901.99,E2 25901.99} C_VEL
LIN {X 0,Y 151.327,Z 1125.543,A -85,B 0,C 180,E1 25911.551,E2 25911.551} C_VEL
LIN {X 0,Y 187.916,Z 1102.9,A -85,B 0,C 180,E1 25917.132,E2 25917.132} C_VEL
LIN {X 0,Y 214.245,Z 1082.562,A -85,B 0,C 180,E1 25920,E2 25920} C_VEL
LIN {X 0,Y 213.488,Z 1083.049,A -85,B 0,C 180,E1 25921.626,E2 25921.626} C_VEL
LIN {X 0,Y 178.239,Z 1108.563,A -85,B 0,C 180,E1 25925.849,E2 25925.849} C_VEL
LIN {X 0,Y 142.546,Z 1128.516,A -85,B 0,C 180,E1 25932.222,E2 25932.222} C_VEL
LIN {X 0,Y 106.94,Z 1143.701,A -85,B 0,C 180,E1 25943.477,E2 25943.477} C_VEL
LIN {X 0,Y 80.326,Z 1152.576,A -85,B 0,C 180,E1 25961.282,E2 25961.282} C_VEL
LIN {X 0,Y 64.75,Z 1156.868,A -85,B 0,C 180,E1 25988.774,E2 25988.774} C_VEL
LIN {X 0,Y 62.898,Z 1157.662,A -85,B 0,C 180,E1 26009.999,E2 26009.999} C_VEL
LIN {X 0,Y 66.608,Z 1156.417,A -85,B 0,C 180,E1 26036.941,E2 26036.941} C_VEL
LIN {X 0,Y 84.982,Z 1151.042,A -85,B 0,C 180,E1 26063.039,E2 26063.039} C_VEL
LIN {X 0,Y 113.148,Z 1141.34,A -85,B 0,C 180,E1 26078.995,E2 26078.995} C_VEL
LIN {X 0,Y 150.44,Z 1124.492,A -85,B 0,C 180,E1 26089.359,E2 26089.359} C_VEL
LIN {X 0,Y 187.978,Z 1102.03,A -85,B 0,C 180,E1 26095.396,E2 26095.396} C_VEL
LIN {X 0,Y 213.485,Z 1082.846,A -85,B 0,C 180,E1 26098.418,E2 26098.418} C_VEL
LIN {X 0,Y 214.219,Z 1082.38,A -85,B 0,C 180,E1 26100,E2 26100} C_VEL
LIN {X 0,Y 194.089,Z 1098.27,A -85,B 0,C 180,E1 26102.173,E2 26102.173} C_VEL
LIN {X 0,Y 179.554,Z 1108.089,A -85,B 0,C 180,E1 26102.594,E2 26102.594} C_VEL
LIN {X 0,Y 164.642,Z 1117.097,A -85,B 0,C 180,E1 26103.123,E2 26103.123} C_VEL
LIN {X 0,Y 127.888,Z 1136.113,A -85,B 0,C 180,E1 26109.863,E2 26109.863} C_VEL
LIN {X 0,Y 93.406,Z 1149.807,A -85,B 0,C 180,E1 26121.733,E2 26121.733} C_VEL
LIN {X 0,Y 65.007,Z 1158.682,A -85,B 0,C 180,E1 26145.863,E2 26145.863} C_VEL
LIN {X 0,Y 55.068,Z 1161.662,A -85,B 0,C 180,E1 26174.098,E2 26174.098} C_VEL
LIN {X 0,Y 54.751,Z 1162.074,A -85,B 0,C 180,E1 26190.002,E2 26190.002} C_VEL
LIN {X 0,Y 58.524,Z 1160.546,A -85,B 0,C 180,E1 26221.045,E2 26221.045} C_VEL
LIN {X 0,Y 78.989,Z 1154.52,A -85,B 0,C 180,E1 26249.283,E2 26249.283} C_VEL
LIN {X 0,Y 112.762,Z 1142.639,A -85,B 0,C 180,E1 26265.984,E2 26265.984} C_VEL
LIN {X 0,Y 148.864,Z 1126.04,A -85,B 0,C 180,E1 26274.417,E2 26274.417} C_VEL
LIN {X 0,Y 186.265,Z 1103.605,A -85,B 0,C 180,E1 26279.486,E2 26279.486} C_VEL
LIN {X 0,Y 199.809,Z 1093.875,A -85,B 0,C 180,E1 26280.787,E2 26280.787} C_VEL
LIN {X 0,Y 160.753,Z 1118.819,A -85,B 0,C 180,E1 26285.537,E2 26285.537} C_VEL
LIN {X 0,Y 123.877,Z 1136.485,A -85,B 0,C 180,E1 26292.957,E2 26292.957} C_VEL
LIN {X 0,Y 85.815,Z 1149.91,A -85,B 0,C 180,E1 26308.449,E2 26308.449} C_VEL
LIN {X 0,Y 66.289,Z 1155.149,A -85,B 0,C 180,E1 26326.926,E2 26326.926} C_VEL
LIN {X 0,Y 55.663,Z 1157.677,A -85,B 0,C 180,E1 26354.269,E2 26354.269} C_VEL
LIN {X 0,Y 54.995,Z 1157.958,A -85,B 0,C 180,E1 26369.998,E2 26369.998} C_VEL
LIN {X 0,Y 59.565,Z 1156.719,A -85,B 0,C 180,E1 26400.441,E2 26400.441} C_VEL
LIN {X 0,Y 80.363,Z 1151.347,A -85,B 0,C 180,E1 26427.669,E2 26427.669} C_VEL
LIN {X 0,Y 113.759,Z 1140.369,A -85,B 0,C 180,E1 26444.016,E2 26444.016} C_VEL
